# B&R Automation Studio project Panasonic_LinkaPowerCP2_A2021055 (part 28)

#### Main.st - Init, cyclic, exit code
```iecst
PROGRAM _INIT
	(* Insert code here *)

END_PROGRAM

PROGRAM _CYCLIC

	//Volanie funkcie SequenceControl//
	SequenceControl(SC:= SC_P3_ZdvizkaPredLeakTestA);

	//Volanie podprogramov//
	OvlZdvizky;

	//Reset sekcie //
	IF P3_ZdvizkaPredLeakTestA.Reset THEN
		SC_P3_ZdvizkaPredLeakTestA.Step:= 0;
		P3_ZdvizkaPredLeakTestA.Reset:= FALSE;
	ELSIF NOT Safety.STAV.Linka_ZonaCS_AKTIVNA THEN
		SC_P3_ZdvizkaPredLeakTestA.Step:= 0;
	END_IF

	CASE SC_P3_ZdvizkaPredLeakTestA.Step OF

		0:
			SC_P3_ZdvizkaPredLeakTestA.StepName:='0 - Nulovanie';
			SC_OvlZdvizky.Step:= 0;
			P3_ZdvizkaPredLeakTestA.Automat:= FALSE;
			P3_ZdvizkaPredLeakTestA.KoniecCyklu:= FALSE;
			P3_ZdvizkaPredLeakTestA.Manual:= FALSE;
			P3_ZdvizkaPredLeakTestA.STAV.PoINIT:= FALSE;
			P3_ZdvizkaPredLeakTestA.OUT.TlmicPaletky_VYSUN:= FALSE;
			P3_Dopravniky.OUT.PriecnyDopravnik1_VPRED:= FALSE;
			P3_ZdvizkaPredLeakTestA.STAV.PrebiehaVyvezeniePaletkyNaTratA:= FALSE;
			P3_ZdvizkaPredLeakTestA.STAV.PrebiehaVyvezeniePaletkyNaTratB:= FALSE;
			P3_HV_Test.STAV.PrebiehaVyvezeniePaletky:= FALSE;

			IF Safety.STAV.Linka_ZonaCS_AKTIVNA AND
				Safety.STAV.P3_ZonaBunky_AKTIVNA AND
				P3_Pracovisko.STAV.HardwareBunky_OK AND
				NOT P3_Pracovisko.STAV.Porucha_ST1 AND
				NOT P3_Pracovisko.STAV.Porucha_ST2 AND
				NOT P3_Pracovisko.STAV.Porucha_ST3 AND
				NOT P3_Pracovisko.STAV.Porucha_ST4 AND
				NOT P3_Pracovisko.STAV.Porucha_ST5 AND
				NOT P3_Pracovisko.STAV.Porucha_ST6 AND
				NOT P3_Pracovisko.STAV.Porucha_ST7 AND
				NOT P3_Pracovisko.STAV.Porucha_ST8 THEN
				SC_P3_ZdvizkaPredLeakTestA.ResetStep:= TRUE;
				SC_P3_ZdvizkaPredLeakTestA.Step:= 1;
			END_IF

		1:
			SC_P3_ZdvizkaPredLeakTestA.StepName:='1 - Cakam na spustenie vyroby';
			P3_ZdvizkaPredLeakTestA.KoniecCyklu:= FALSE;
			IF P3_ZdvizkaPredLeakTestA.Automat THEN
				SC_P3_ZdvizkaPredLeakTestA.Step:= 2;
			ELSIF P3_ZdvizkaPredLeakTestA.Manual THEN
				SC_P3_ZdvizkaPredLeakTestA.Step:= 700;
			END_IF

			//********************************************************Inicializácia****************************************************************************//

		2:
			SC_P3_ZdvizkaPredLeakTestA.StepName:='2 - Inicializacia - cakam na spustenie inicializacie';
			SC_P3_ZdvizkaPredLeakTestA.IdleTime.PT:= T#500ms;
			SC_P3_ZdvizkaPredLeakTestA.AlarmTime.PT:= T#5s;

			IF P3_Dopravniky.STAV.PoINIT AND P3_ZdvizkaPredLeakTestB.STAV.PoINIT THEN
				SC_P3_ZdvizkaPredLeakTestA.ResetStep:= TRUE;
				SC_P3_ZdvizkaPredLeakTestA.Step:= 5;
			END_IF

		5:
			SC_P3_ZdvizkaPredLeakTestA.StepName:='5 - Inicializacia - kontrola pozicie zdvizky';
			SC_P3_ZdvizkaPredLeakTestA.IdleTime.PT:= T#500ms;
			SC_P3_ZdvizkaPredLeakTestA.AlarmTime.PT:= T#5s;

			IF P3_ZdvizkaPredLeakTestA.IN.Zdvizka_StrednaPoloha AND P3_ZdvizkaPredLeakTestA.IN.PritomnostPaletky THEN
				P3_ZdvizkaPredLeakTestA.STAV.PoINIT:= TRUE;
				SC_P3_ZdvizkaPredLeakTestA.ResetStep:= TRUE;
				SC_P3_ZdvizkaPredLeakTestA.Step:= 100;
			ELSIF P3_ZdvizkaPredLeakTestA.IN.Zdvizka_StrednaPoloha AND NOT P3_ZdvizkaPredLeakTestA.IN.PritomnostPaletky THEN
				SC_P3_ZdvizkaPredLeakTestA.ResetStep:= TRUE;
				SC_P3_ZdvizkaPredLeakTestA.Step:= 6;
			ELSE
				SC_P3_ZdvizkaPredLeakTestA.ResetStep:= TRUE;
				SC_P3_ZdvizkaPredLeakTestA.Step:= 8;
			END_IF

		6:
			SC_P3_ZdvizkaPredLeakTestA.StepName:='5 - Inicializacia - vysunutie tlmica';
			SC_P3_ZdvizkaPredLeakTestA.IdleTime.PT:= T#500ms;
			SC_P3_ZdvizkaPredLeakTestA.AlarmTime.PT:= T#5s;

			IF NOT SC_P3_ZdvizkaPredLeakTestA.Switch1 THEN
				P3_ZdvizkaPredLeakTestA.OUT.TlmicPaletky_VYSUN:= TRUE;
				SC_P3_ZdvizkaPredLeakTestA.IdleTime.IN:= TRUE;
				SC_P3_ZdvizkaPredLeakTestA.Switch1:= TRUE;
			END_IF

			IF SC_P3_ZdvizkaPredLeakTestA.IdleTime.Q THEN
				P3_ZdvizkaPredLeakTestA.OUT.TlmicPaletky_VYSUN:= FALSE;
				P3_ZdvizkaPredLeakTestA.STAV.PoINIT:= TRUE;
				SC_P3_ZdvizkaPredLeakTestA.ResetStep:= TRUE;
				SC_P3_ZdvizkaPredLeakTestA.Step:= 100;
			END_IF

		8:
			SC_P3_ZdvizkaPredLeakTestA.StepName:='8 - Inicializacia - presun zdvizky do strednej polohy';
			SC_P3_ZdvizkaPredLeakTestA.IdleTime.PT:= T#5s;
			SC_P3_ZdvizkaPredLeakTestA.AlarmTime.PT:= T#5s;

			IF NOT SC_P3_ZdvizkaPredLeakTestA.Switch1 AND SC_OvlZdvizky.Step = 1 THEN
				Zdvizku_VYSTRED:= TRUE;
				SC_P3_ZdvizkaPredLeakTestA.Switch1:= TRUE;
			END_IF

			IF P3_ZdvizkaPredLeakTestA.IN.Zdvizka_StrednaPoloha THEN
				SC_P3_ZdvizkaPredLeakTestA.ResetStep:= TRUE;
				SC_P3_ZdvizkaPredLeakTestA.Step:= 10;
			END_IF

		10:
			SC_P3_ZdvizkaPredLeakTestA.StepName:='10 - Inicializacia - hladania paletky';
			SC_P3_ZdvizkaPredLeakTestA.IdleTime.PT:= T#5s;
			SC_P3_ZdvizkaPredLeakTestA.AlarmTime.PT:= T#5s;

			SC_P3_ZdvizkaPredLeakTestA.IdleTime.IN:= TRUE;

			IF SC_P3_ZdvizkaPredLeakTestA.IdleTime.Q THEN
				SC_P3_ZdvizkaPredLeakTestA.ResetStep:= TRUE;
				SC_P3_ZdvizkaPredLeakTestA.Step:= 5;
			END_IF

			//********************************************************Automatický režim****************************************************************************//

		100:
			SC_P3_ZdvizkaPredLeakTestA.StepName:='100 - Automaticky Rezim - cakam na príchod paletky na zdvizku';
			SC_P3_ZdvizkaPredLeakTestA.IdleTime.PT:= T#700ms;
			SC_P3_ZdvizkaPredLeakTestA.AlarmTime.PT:= T#5s;

			SC_P3_ZdvizkaPredLeakTestA.IdleTime.IN:= P3_ZdvizkaPredLeakTestA.IN.PritomnostPaletky;

			IF P3_ZdvizkaPredLeakTestA.IN.PritomnostPaletky THEN
				P3_HV_Test.STAV.PrebiehaVyvezeniePaletky:= FALSE;
			END_IF

			IF P3_ZdvizkaPredLeakTestA.KoniecCyklu AND NOT P3_HV_Test.Automat THEN
				SC_P3_ZdvizkaPredLeakTestA.ResetStep:= TRUE;
				SC_P3_ZdvizkaPredLeakTestA.Step:= 0;
			ELSIF SC_P3_ZdvizkaPredLeakTestA.IdleTime.Q THEN
				SC_P3_ZdvizkaPredLeakTestA.ResetStep:= TRUE;
				SC_P3_ZdvizkaPredLeakTestA.Step:= 101;
			END_IF

		101:
			SC_P3_ZdvizkaPredLeakTestA.StepName:='101 - Automaticky Rezim - rozhodnutie o smere vyvazania';
			SC_P3_ZdvizkaPredLeakTestA.IdleTime.PT:= T#200ms;
			SC_P3_ZdvizkaPredLeakTestA.AlarmTime.PT:= T#5s;

			IF P3_ZdvizkaPredLeakTestA.KoniecCyklu AND NOT P3_HV_Test.Automat THEN
				SC_P3_ZdvizkaPredLeakTestA.ResetStep:= TRUE;
				SC_P3_ZdvizkaPredLeakTestA.Step:= 0;
			ELSIF P3_LeakageTestA.STAV.Tester_ON AND NOT P3_LeakageTestA.RFID_hlava.PritomnostPaletky AND SC_P3_LeakageTestA.Step = 100 AND NOT P3_ZdvizkaPredLeakTestA.STAV.PrebiehaVyvezeniePaletkyNaTratA THEN
				SC_P3_ZdvizkaPredLeakTestA.ResetStep:= TRUE;
				SC_P3_ZdvizkaPredLeakTestA.Step:= 110;
			ELSIF P3_LeakageTestB.STAV.Tester_ON AND NOT P3_ZdvizkaPredLeakTestB.IN.PritomnostPaletky AND NOT P3_LeakageTestB.RFID_hlava.PritomnostPaletky AND SC_P3_ZdvizkaPredLeakTestB.Step = 100 AND NOT P3_ZdvizkaPredLeakTestA.STAV.PrebiehaVyvezeniePaletkyNaTratB THEN
				SC_P3_ZdvizkaPredLeakTestA.ResetStep:= TRUE;
				SC_P3_ZdvizkaPredLeakTestA.Step:= 120;
			END_IF

			//Vyvážanie na trať A//

		110:
			SC_P3_ZdvizkaPredLeakTestA.StepName:='110 - Automaticky Rezim - presun zdvizky do spodnej polohy';
			SC_P3_ZdvizkaPredLeakTestA.IdleTime.PT:= T#200ms;
			SC_P3_ZdvizkaPredLeakTestA.AlarmTime.PT:= T#5s;

			IF NOT SC_P3_ZdvizkaPredLeakTestA.Switch1 AND SC_OvlZdvizky.Step = 1 THEN
				Zdvizku_ZASUN:= TRUE;
				P3_ZdvizkaPredLeakTestA.STAV.PrebiehaVyvezeniePaletkyNaTratA:= TRUE;
				SC_P3_ZdvizkaPredLeakTestA.Switch1:= TRUE;
			END_IF

			IF P3_ZdvizkaPredLeakTestA.IN.Zdvizka_SpodnaPoloha THEN
				SC_P3_ZdvizkaPredLeakTestA.ResetStep:= TRUE;
				SC_P3_ZdvizkaPredLeakTestA.Step:= 113;
			END_IF

		113:
			SC_P3_ZdvizkaPredLeakTestA.StepName:='113 - Automaticky Rezim - cakam na ukoncenie vyvazania na Trat A';
			SC_P3_ZdvizkaPredLeakTestA.IdleTime.PT:= T#500ms;
			SC_P3_ZdvizkaPredLeakTestA.AlarmTime.PT:= T#5s;

			IF P3_LeakageTestA.RFID_hlava.PritomnostPaletky AND SC_OvlZdvizky.Step = 1 AND NOT SC_P3_ZdvizkaPredLeakTestA.Switch1 THEN
				Zdvizku_VYSTRED:= TRUE;
				SC_P3_ZdvizkaPredLeakTestA.Switch1:= TRUE;
			END_IF

			IF P3_ZdvizkaPredLeakTestA.IN.Zdvizka_StrednaPoloha THEN
				SC_P3_ZdvizkaPredLeakTestA.ResetStep:= TRUE;
				SC_P3_ZdvizkaPredLeakTestA.Step:= 130;
			END_IF

			//Vyvážanie na trať B//

		120:
			SC_P3_ZdvizkaPredLeakTestA.StepName:='120 - Automaticky Rezim - presun zdviziek do hornej polohy';
			SC_P3_ZdvizkaPredLeakTestA.IdleTime.PT:= T#200ms;
			SC_P3_ZdvizkaPredLeakTestA.AlarmTime.PT:= T#5s;

			IF NOT SC_P3_ZdvizkaPredLeakTestA.Switch1 AND SC_OvlZdvizky.Step = 1 THEN
				Zdvizku_VYSUN:= TRUE;
				P3_ZdvizkaPredLeakTestB.OUT.Zdvizku_ZASUN:= FALSE;
				P3_ZdvizkaPredLeakTestB.OUT.Zdvizku_VYSUN:= TRUE;
				P3_ZdvizkaPredLeakTestA.STAV.PrebiehaVyvezeniePaletkyNaTratB:= TRUE;
				SC_P3_ZdvizkaPredLeakTestA.Switch1:= TRUE;
			END_IF

			IF P3_ZdvizkaPredLeakTestA.IN.Zdvizka_HornaPoloha AND P3_ZdvizkaPredLeakTestB.IN.Zdvizka_HornaPoloha THEN
				SC_P3_ZdvizkaPredLeakTestA.ResetStep:= TRUE;
				SC_P3_ZdvizkaPredLeakTestA.Step:= 123;
			END_IF

		123:
			SC_P3_ZdvizkaPredLeakTestA.StepName:='123 - Automaticky Rezim - cakam na ukoncenie vyvazania na Trat B';
			SC_P3_ZdvizkaPredLeakTestA.IdleTime.PT:= T#500ms;
			SC_P3_ZdvizkaPredLeakTestA.AlarmTime.PT:= T#5s;

			SC_P3_ZdvizkaPredLeakTestA.IdleTime.IN:= P3_ZdvizkaPredLeakTestB.IN.PritomnostPaletky;

			IF NOT SC_P3_ZdvizkaPredLeakTestA.Switch1 THEN
				P3_Dopravniky.OUT.PriecnyDopravnik1_VPRED:= TRUE;
				SC_P3_ZdvizkaPredLeakTestA.Switch1:= TRUE;
			END_IF

			IF SC_P3_ZdvizkaPredLeakTestA.IdleTime.Q THEN
				P3_Dopravniky.OUT.PriecnyDopravnik1_VPRED:= FALSE;
				SC_P3_ZdvizkaPredLeakTestA.ResetStep:= TRUE;
				SC_P3_ZdvizkaPredLeakTestA.Step:= 125;
			END_IF

		125:
			SC_P3_ZdvizkaPredLeakTestA.StepName:='123 - Automaticky Rezim - cakam na presun zdviziek do strednej polohy';
			SC_P3_ZdvizkaPredLeakTestA.IdleTime.PT:= T#1s;
			SC_P3_ZdvizkaPredLeakTestA.AlarmTime.PT:= T#5s;

			IF NOT SC_P3_ZdvizkaPredLeakTestA.Switch1 AND SC_OvlZdvizky.Step = 1 THEN
				Zdvizku_VYSTRED:= TRUE;
				P3_ZdvizkaPredLeakTestB.OUT.Zdvizku_ZASUN:= FALSE;
				P3_ZdvizkaPredLeakTestB.OUT.Zdvizku_VYSUN:= FALSE;
				SC_P3_ZdvizkaPredLeakTestA.Switch1:= TRUE;
			END_IF

			IF P3_ZdvizkaPredLeakTestA.IN.Zdvizka_StrednaPoloha AND P3_ZdvizkaPredLeakTestB.IN.Zdvizka_StrednaPoloha THEN
				P3_ZdvizkaPredLeakTestA.STAV.PrebiehaVyvezeniePaletkyNaTratB:= FALSE;
				SC_P3_ZdvizkaPredLeakTestA.ResetStep:= TRUE;
				SC_P3_ZdvizkaPredLeakTestA.Step:= 130;
			END_IF

			//Vysunutie tlmenia paletky//

		130:
			SC_P3_ZdvizkaPredLeakTestA.StepName:='130 - Automaticky Rezim - vysunutie tlamena paletky';
			SC_P3_ZdvizkaPredLeakTestA.IdleTime.PT:= T#1s;
			SC_P3_ZdvizkaPredLeakTestA.AlarmTime.PT:= T#5s;

			IF NOT SC_P3_ZdvizkaPredLeakTestA.Switch1 THEN
				P3_ZdvizkaPredLeakTestA.OUT.TlmicPaletky_VYSUN:= TRUE;
				SC_P3_ZdvizkaPredLeakTestA.IdleTime.IN:= TRUE;
				SC_P3_ZdvizkaPredLeakTestA.Switch1:= TRUE;
			END_IF

			IF SC_P3_ZdvizkaPredLeakTestA.IdleTime.Q THEN
				P3_ZdvizkaPredLeakTestA.OUT.TlmicPaletky_VYSUN:= FALSE;
				SC_P3_ZdvizkaPredLeakTestA.ResetStep:= TRUE;
				SC_P3_ZdvizkaPredLeakTestA.Step:= 100;
			END_IF

			//*******************************************************Manuálny režim*******************************************************************************//
		700:
			SC_P3_ZdvizkaPredLeakTestA.StepName:='700 - Manualny Rezim';
			SC_P3_ZdvizkaPredLeakTestA.IdleTime.PT:= T#8s;
			SC_P3_ZdvizkaPredLeakTestA.AlarmTime.PT:= T#5s;

	END_CASE

				END_PROGRAM

PROGRAM _EXIT
				(* Insert code here *)

				END_PROGRAM
```

#### Variables.var - Local variables
```iecst
VAR
	SC_OvlZdvizky : SequenceControlTyp;
	Zdvizku_VYSUN : BOOL;
	Zdvizku_ZASUN : BOOL;
	Zdvizku_VYSTRED : BOOL := FALSE;
END_VAR
```

#### OvlZdvizky.st
```iecst
ACTION OvlZdvizky:

	//Volanie funkcie SequenceControl//
	SequenceControl(SC:= SC_OvlZdvizky);

	CASE SC_OvlZdvizky.Step OF

		0:
			SC_OvlZdvizky.StepName:= '0 - Nulovanie';
			Zdvizku_VYSUN:= FALSE;
			Zdvizku_ZASUN:= FALSE;
			Zdvizku_VYSTRED:= FALSE;

			IF SC_P3_ZdvizkaPredLeakTestA.Step <> 0 THEN
				SC_OvlZdvizky.ResetStep:= TRUE;
				SC_OvlZdvizky.Step:= 1;
			END_IF

		1:
			SC_OvlZdvizky.StepName:= '1 - Rozhodnutie o cinnosti';
			IF Zdvizku_VYSUN THEN
				SC_OvlZdvizky.Step:= 10;
			ELSIF Zdvizku_ZASUN THEN
				SC_OvlZdvizky.Step:= 20;
			ELSIF Zdvizku_VYSTRED THEN
				SC_OvlZdvizky.Step:= 30;
			END_IF

		10:
			SC_OvlZdvizky.StepName:= '10 - Vysunutie zdvizky hore';
			SC_OvlZdvizky.IdleTime.PT:= T#3s;
			SC_OvlZdvizky.AlarmTime.PT:= T#6s;

			IF P3_ZdvizkaPredLeakTestA.Automat THEN
				SC_OvlZdvizky.AlarmTime.IN:= TRUE;
			ELSE
				SC_OvlZdvizky.IdleTime.IN:= TRUE;
			END_IF

			IF NOT SC_OvlZdvizky.Switch1 THEN
				P3_ZdvizkaPredLeakTestA.OUT.Zdvizku_ZASUN:= FALSE;
				P3_ZdvizkaPredLeakTestA.OUT.Zdvizku_VYSUN:= TRUE;
				SC_OvlZdvizky.Switch1:= TRUE;
			END_IF

			IF P3_ZdvizkaPredLeakTestA.IN.Zdvizka_HornaPoloha OR SC_OvlZdvizky.IdleTime.Q THEN
				SC_OvlZdvizky.ResetStep:= TRUE;
				SC_OvlZdvizky.Step:= 0;
			ELSIF SC_OvlZdvizky.AlarmTime.Q THEN
				P34_Alarmy[368]:= TRUE;
				P3_Pracovisko.STAV.Porucha_ST3:= TRUE;
			END_IF

		20:
			SC_OvlZdvizky.StepName:= '20 - Zasunutie zdvizky dole';
			SC_OvlZdvizky.IdleTime.PT:= T#3s;
			SC_OvlZdvizky.AlarmTime.PT:= T#6s;

			IF P3_ZdvizkaPredLeakTestA.Automat THEN
				SC_OvlZdvizky.AlarmTime.IN:= TRUE;
			ELSE
				SC_OvlZdvizky.IdleTime.IN:= TRUE;
			END_IF

			IF NOT SC_OvlZdvizky.Switch1 THEN
				P3_ZdvizkaPredLeakTestA.OUT.Zdvizku_VYSUN:= FALSE;
				P3_ZdvizkaPredLeakTestA.OUT.Zdvizku_ZASUN:= TRUE;
				SC_OvlZdvizky.Switch1:= TRUE;
			END_IF

			IF P3_ZdvizkaPredLeakTestA.IN.Zdvizka_SpodnaPoloha OR SC_OvlZdvizky.IdleTime.Q THEN
				SC_OvlZdvizky.ResetStep:= TRUE;
				SC_OvlZdvizky.Step:= 0;
			ELSIF SC_OvlZdvizky.AlarmTime.Q THEN
				P34_Alarmy[369]:= TRUE;
				P3_Pracovisko.STAV.Porucha_ST3:= TRUE;
			END_IF

		30:
			SC_OvlZdvizky.StepName:= '30 - Presun zdvizky do strednej polohy';
			SC_OvlZdvizky.IdleTime.PT:= T#3s;
			SC_OvlZdvizky.AlarmTime.PT:= T#6s;

			IF P3_ZdvizkaPredLeakTestA.Automat THEN
				SC_OvlZdvizky.AlarmTime.IN:= TRUE;
			ELSE
				SC_OvlZdvizky.IdleTime.IN:= TRUE;
			END_IF

			IF NOT SC_OvlZdvizky.Switch1 THEN
				P3_ZdvizkaPredLeakTestA.OUT.Zdvizku_VYSUN:= FALSE;
				P3_ZdvizkaPredLeakTestA.OUT.Zdvizku_ZASUN:= FALSE;
				SC_OvlZdvizky.Switch1:= TRUE;
			END_IF

			IF P3_ZdvizkaPredLeakTestA.IN.Zdvizka_StrednaPoloha OR SC_OvlZdvizky.IdleTime.Q THEN
				SC_OvlZdvizky.ResetStep:= TRUE;
				SC_OvlZdvizky.Step:= 0;
			ELSIF SC_OvlZdvizky.AlarmTime.Q THEN
				P34_Alarmy[370]:= TRUE;
				P3_Pracovisko.STAV.Porucha_ST3:= TRUE;
			END_IF

	END_CASE

END_ACTION
```

### Program Logical/Program/Pracovisko_3/P3_ZdvizkaPredLeakTestB (IEC)

#### Main.st - Init, cyclic, exit code
```iecst
PROGRAM _INIT
	(* Insert code here *)

END_PROGRAM

PROGRAM _CYCLIC

	//Volanie funkcie SequenceControl//
	SequenceControl(SC:= SC_P3_ZdvizkaPredLeakTestB);

	//Volanie podprogramov//
	OvlZdvizky;

	//Reset sekcie //
	IF P3_ZdvizkaPredLeakTestB.Reset THEN
		SC_P3_ZdvizkaPredLeakTestB.Step:= 0;
		P3_ZdvizkaPredLeakTestB.Reset:= FALSE;
	ELSIF NOT Safety.STAV.Linka_ZonaCS_AKTIVNA THEN
		SC_P3_ZdvizkaPredLeakTestB.Step:= 0;
	END_IF

	CASE SC_P3_ZdvizkaPredLeakTestB.Step OF

		0:
			SC_P3_ZdvizkaPredLeakTestB.StepName:='0 - Nulovanie';
			SC_OvlZdvizky.Step:= 0;
			P3_ZdvizkaPredLeakTestB.Automat:= FALSE;
			P3_ZdvizkaPredLeakTestB.KoniecCyklu:= FALSE;
			P3_ZdvizkaPredLeakTestB.Manual:= FALSE;
			P3_ZdvizkaPredLeakTestB.STAV.PoINIT:= FALSE;
			P3_Dopravniky.OUT.PriecnyDopravnik1_VPRED:= FALSE;
			P3_ZdvizkaPredLeakTestB.STAV.PrebiehaVyvezeniePaletky:= FALSE;
			P3_ZdvizkaPredLeakTestA.STAV.PrebiehaVyvezeniePaletkyNaTratB:= FALSE;

			IF Safety.STAV.Linka_ZonaCS_AKTIVNA AND
				Safety.STAV.P3_ZonaBunky_AKTIVNA AND
				P3_Pracovisko.STAV.HardwareBunky_OK AND
				NOT P3_Pracovisko.STAV.Porucha_ST1 AND
				NOT P3_Pracovisko.STAV.Porucha_ST2 AND
				NOT P3_Pracovisko.STAV.Porucha_ST3 AND
				NOT P3_Pracovisko.STAV.Porucha_ST4 AND
				NOT P3_Pracovisko.STAV.Porucha_ST5 AND
				NOT P3_Pracovisko.STAV.Porucha_ST6 AND
				NOT P3_Pracovisko.STAV.Porucha_ST7 AND
				NOT P3_Pracovisko.STAV.Porucha_ST8 THEN
				SC_P3_ZdvizkaPredLeakTestB.ResetStep:= TRUE;
				SC_P3_ZdvizkaPredLeakTestB.Step:= 1;
			END_IF

		1:
			SC_P3_ZdvizkaPredLeakTestB.StepName:='1 - Cakam na spustenie vyroby';
			P3_ZdvizkaPredLeakTestB.KoniecCyklu:= FALSE;
			IF P3_ZdvizkaPredLeakTestB.Automat THEN
				SC_P3_ZdvizkaPredLeakTestB.Step:= 2;
			ELSIF P3_ZdvizkaPredLeakTestB.Manual THEN
				SC_P3_ZdvizkaPredLeakTestB.Step:= 700;
			END_IF

			//********************************************************Inicializácia****************************************************************************//

		2:
			SC_P3_ZdvizkaPredLeakTestB.StepName:='2 - Inicializacia - cakam na spustenie inicializacie';
			SC_P3_ZdvizkaPredLeakTestB.IdleTime.PT:= T#500ms;
			SC_P3_ZdvizkaPredLeakTestB.AlarmTime.PT:= T#5s;

			IF P3_Dopravniky.STAV.PoINIT THEN
				SC_P3_ZdvizkaPredLeakTestB.ResetStep:= TRUE;
				SC_P3_ZdvizkaPredLeakTestB.Step:= 5;
			END_IF

		5:
			SC_P3_ZdvizkaPredLeakTestB.StepName:='5 - Inicializacia - kontrola pozicie zdvizky';
			SC_P3_ZdvizkaPredLeakTestB.IdleTime.PT:= T#500ms;
			SC_P3_ZdvizkaPredLeakTestB.AlarmTime.PT:= T#5s;

			IF P3_ZdvizkaPredLeakTestB.IN.Zdvizka_StrednaPoloha AND P3_ZdvizkaPredLeakTestB.IN.PritomnostPaletky THEN
				P3_ZdvizkaPredLeakTestB.STAV.PoINIT:= TRUE;
				SC_P3_ZdvizkaPredLeakTestB.ResetStep:= TRUE;
				SC_P3_ZdvizkaPredLeakTestB.Step:= 120;
			ELSE
				SC_P3_ZdvizkaPredLeakTestB.ResetStep:= TRUE;
				SC_P3_ZdvizkaPredLeakTestB.Step:= 8;
			END_IF

		8:
			SC_P3_ZdvizkaPredLeakTestB.StepName:='8 - Inicializacia - presun zdvizky do hornej polohy';
			SC_P3_ZdvizkaPredLeakTestB.IdleTime.PT:= T#500ms;
			SC_P3_ZdvizkaPredLeakTestB.AlarmTime.PT:= T#5s;

			IF NOT SC_P3_ZdvizkaPredLeakTestB.Switch1 AND SC_OvlZdvizky.Step = 1 THEN
				Zdvizku_VYSUN:= TRUE;
				SC_P3_ZdvizkaPredLeakTestB.Switch1:= TRUE;
			END_IF

			IF P3_ZdvizkaPredLeakTestB.IN.Zdvizka_HornaPoloha THEN
				SC_P3_ZdvizkaPredLeakTestB.ResetStep:= TRUE;
				SC_P3_ZdvizkaPredLeakTestB.Step:= 10;
			END_IF

		10:
			SC_P3_ZdvizkaPredLeakTestB.StepName:='10 - Inicializacia - kontrola pritomnosti paletky na zdvizke pred Leakage Testom A';
			SC_P3_ZdvizkaPredLeakTestB.IdleTime.PT:= T#500ms;
			SC_P3_ZdvizkaPredLeakTestB.AlarmTime.PT:= T#5s;

			IF NOT P3_ZdvizkaPredLeakTestA.IN.PritomnostPaletky THEN
				P3_ZdvizkaPredLeakTestA.OUT.Zdvizku_ZASUN:= FALSE;
				P3_ZdvizkaPredLeakTestA.OUT.Zdvizku_VYSUN:= TRUE;
				SC_P3_ZdvizkaPredLeakTestB.ResetStep:= TRUE;
				SC_P3_ZdvizkaPredLeakTestB.Step:= 11;
			ELSE
				SC_P3_ZdvizkaPredLeakTestB.ResetStep:= TRUE;
				SC_P3_ZdvizkaPredLeakTestB.Step:= 13;
			END_IF

		11:
			SC_P3_ZdvizkaPredLeakTestB.StepName:='11 - Inicializacia - cakam na zodvihnutie zdvizky Pred Leakage Testom A';
			SC_P3_ZdvizkaPredLeakTestB.IdleTime.PT:= T#500ms;
			SC_P3_ZdvizkaPredLeakTestB.AlarmTime.PT:= T#5s;

			IF P3_ZdvizkaPredLeakTestA.IN.Zdvizka_HornaPoloha THEN
				SC_P3_ZdvizkaPredLeakTestB.ResetStep:= TRUE;
				SC_P3_ZdvizkaPredLeakTestB.Step:= 13;
			END_IF

		13:
			SC_P3_ZdvizkaPredLeakTestB.StepName:='13 - Inicializacia - spustenie priecneho dopravnika';
			SC_P3_ZdvizkaPredLeakTestB.IdleTime.PT:= T#500ms;
			SC_P3_ZdvizkaPredLeakTestB.AlarmTime.PT:= T#7s;

			SC_P3_ZdvizkaPredLeakTestB.IdleTime.IN:= P3_ZdvizkaPredLeakTestB.IN.PritomnostPaletky AND P3_ZdvizkaPredLeakTestB.IN.PoziciaPaletky_OK;

			IF NOT SC_P3_ZdvizkaPredLeakTestB.Switch1 THEN
				P3_Dopravniky.OUT.PriecnyDopravnik1_VPRED:= TRUE;
				SC_P3_ZdvizkaPredLeakTestB.AlarmTime.IN:= TRUE;
				SC_P3_ZdvizkaPredLeakTestB.Switch1:= TRUE;
			END_IF

			IF SC_P3_ZdvizkaPredLeakTestB.IdleTime.Q THEN
				P3_Dopravniky.OUT.PriecnyDopravnik1_VPRED:= FALSE;
				SC_P3_ZdvizkaPredLeakTestB.ResetStep:= TRUE;
				SC_P3_ZdvizkaPredLeakTestB.Step:= 15;
			ELSIF SC_P3_ZdvizkaPredLeakTestB.AlarmTime.Q THEN
				P3_Dopravniky.OUT.PriecnyDopravnik1_VPRED:= FALSE;
				SC_P3_ZdvizkaPredLeakTestB.ResetStep:= TRUE;
				SC_P3_ZdvizkaPredLeakTestB.Step:= 15;
			END_IF

		15:
			SC_P3_ZdvizkaPredLeakTestB.StepName:='15 - Inicializacia - presun zdvizky do strednej polohy';
			SC_P3_ZdvizkaPredLeakTestB.IdleTime.PT:= T#500ms;
			SC_P3_ZdvizkaPredLeakTestB.AlarmTime.PT:= T#5s;

			IF NOT SC_P3_ZdvizkaPredLeakTestB.Switch1 AND SC_OvlZdvizky.Step = 1 THEN
				Zdvizku_VYSTRED:= TRUE;
				P3_ZdvizkaPredLeakTestA.OUT.Zdvizku_ZASUN:= FALSE;
				P3_ZdvizkaPredLeakTestA.OUT.Zdvizku_VYSUN:= FALSE;
				SC_P3_ZdvizkaPredLeakTestB.Switch1:= TRUE;
			END_IF

			IF P3_ZdvizkaPredLeakTestB.IN.Zdvizka_StrednaPoloha AND P3_ZdvizkaPredLeakTestA.IN.Zdvizka_StrednaPoloha THEN
				P3_ZdvizkaPredLeakTestB.STAV.PoINIT:= TRUE;
				IF P3_ZdvizkaPredLeakTestB.IN.PritomnostPaletky THEN
					SC_P3_ZdvizkaPredLeakTestB.ResetStep:= TRUE;
					SC_P3_ZdvizkaPredLeakTestB.Step:= 120;
				ELSE
					SC_P3_ZdvizkaPredLeakTestB.ResetStep:= TRUE;
					SC_P3_ZdvizkaPredLeakTestB.Step:= 100;
				END_IF
			END_IF

		//********************************************************Automatický režim****************************************************************************//
		100:
			SC_P3_ZdvizkaPredLeakTestB.StepName:='100 - Automaticky Rezim - cakam na prichod paletky na zdvizku';
			SC_P3_ZdvizkaPredLeakTestB.IdleTime.PT:= T#200ms;
			SC_P3_ZdvizkaPredLeakTestB.AlarmTime.PT:= T#5s;

			SC_P3_ZdvizkaPredLeakTestB.IdleTime.IN:= P3_ZdvizkaPredLeakTestB.IN.PritomnostPaletky AND P3_ZdvizkaPredLeakTestB.IN.Zdvizka_StrednaPoloha;

			IF P3_ZdvizkaPredLeakTestB.IN.PritomnostPaletky THEN
				P3_ZdvizkaPredLeakTestA.STAV.PrebiehaVyvezeniePaletkyNaTratB:= FALSE;
			END_IF

			IF P3_ZdvizkaPredLeakTestB.KoniecCyklu AND NOT P3_ZdvizkaPredLeakTestA.Automat THEN
				SC_P3_ZdvizkaPredLeakTestB.ResetStep:= TRUE;
				SC_P3_ZdvizkaPredLeakTestB.Step:= 0;
			ELSIF SC_P3_ZdvizkaPredLeakTestB.IdleTime.Q THEN
				SC_P3_ZdvizkaPredLeakTestB.ResetStep:= TRUE;
				SC_P3_ZdvizkaPredLeakTestB.Step:= 120;
			END_IF

		120:
			SC_P3_ZdvizkaPredLeakTestB.StepName:='120 - Automaticky Rezim - cakam na vyvezenie na stoper Leakage Testu B';
			SC_P3_ZdvizkaPredLeakTestB.IdleTime.PT:= T#500ms;
			SC_P3_ZdvizkaPredLeakTestB.AlarmTime.PT:= T#5s;

			IF P3_ZdvizkaPredLeakTestB.KoniecCyklu AND NOT P3_ZdvizkaPredLeakTestA.Automat THEN
				SC_P3_ZdvizkaPredLeakTestB.ResetStep:= TRUE;
				SC_P3_ZdvizkaPredLeakTestB.Step:= 0;
			ELSIF NOT P3_LeakageTestB.RFID_hlava.PritomnostPaletky AND SC_P3_LeakageTestB.Step = 100 THEN
				SC_P3_ZdvizkaPredLeakTestB.ResetStep:= TRUE;
				SC_P3_ZdvizkaPredLeakTestB.Step:= 123;
			END_IF

		123:
			SC_P3_ZdvizkaPredLeakTestB.StepName:='123 - Automaticky Rezim - presun zdvizky do spodnej polohy';
			SC_P3_ZdvizkaPredLeakTestB.IdleTime.PT:= T#200ms;
			SC_P3_ZdvizkaPredLeakTestB.AlarmTime.PT:= T#5s;

			IF NOT SC_P3_ZdvizkaPredLeakTestB.Switch1 AND SC_OvlZdvizky.Step = 1 THEN
				Zdvizku_ZASUN:= TRUE;
				P3_ZdvizkaPredLeakTestB.STAV.PrebiehaVyvezeniePaletky:= TRUE;
				SC_P3_ZdvizkaPredLeakTestB.Switch1:= TRUE;
			END_IF

			IF P3_ZdvizkaPredLeakTestB.IN.Zdvizka_SpodnaPoloha THEN
				SC_P3_ZdvizkaPredLeakTestB.ResetStep:= TRUE;
				SC_P3_ZdvizkaPredLeakTestB.Step:= 125;
			END_IF

		125:
			SC_P3_ZdvizkaPredLeakTestB.StepName:='125 - Automaticky Rezim - cakam na ukoncenie vyvazania na stoper Leakage Testu B';
			SC_P3_ZdvizkaPredLeakTestB.IdleTime.PT:= T#500ms;
			SC_P3_ZdvizkaPredLeakTestB.AlarmTime.PT:= T#5s;

			IF P3_LeakageTestB.RFID_hlava.PritomnostPaletky AND NOT SC_P3_ZdvizkaPredLeakTestB.Switch1 AND SC_OvlZdvizky.Step = 1 THEN
				Zdvizku_VYSTRED:= TRUE;
				SC_P3_ZdvizkaPredLeakTestB.Switch1:= TRUE;
			END_IF

			IF P3_ZdvizkaPredLeakTestB.IN.Zdvizka_StrednaPoloha THEN
				SC_P3_ZdvizkaPredLeakTestB.ResetStep:= TRUE;
				SC_P3_ZdvizkaPredLeakTestB.Step:= 100;
			END_IF

			//*******************************************************Manuálny režim*******************************************************************************//
		700:
			SC_P3_ZdvizkaPredLeakTestB.StepName:='700 - Manualny Rezim';
			SC_P3_ZdvizkaPredLeakTestB.IdleTime.PT:= T#8s;
			SC_P3_ZdvizkaPredLeakTestB.AlarmTime.PT:= T#5s;

	END_CASE

	END_PROGRAM

PROGRAM _EXIT
						(* Insert code here *)

						END_PROGRAM
```

#### Variables.var - Local variables
```iecst
VAR
	SC_OvlZdvizky : SequenceControlTyp;
	Zdvizku_VYSUN : BOOL;
	Zdvizku_ZASUN : BOOL;
	Zdvizku_VYSTRED : BOOL := FALSE;
END_VAR
```

#### OvlZdvizky.st
```iecst
ACTION OvlZdvizky:

	//Volanie funkcie SequenceControl//
	SequenceControl(SC:= SC_OvlZdvizky);

	CASE SC_OvlZdvizky.Step OF

		0:
			SC_OvlZdvizky.StepName:= '0 - Nulovanie';
			Zdvizku_VYSUN:= FALSE;
			Zdvizku_ZASUN:= FALSE;
			Zdvizku_VYSTRED:= FALSE;

			IF SC_P3_ZdvizkaPredLeakTestB.Step <> 0 THEN
				SC_OvlZdvizky.ResetStep:= TRUE;
				SC_OvlZdvizky.Step:= 1;
			END_IF

		1:
			SC_OvlZdvizky.StepName:= '1 - Rozhodnutie o cinnosti';
			IF Zdvizku_VYSUN THEN
				SC_OvlZdvizky.Step:= 10;
			ELSIF Zdvizku_ZASUN THEN
				SC_OvlZdvizky.Step:= 20;
			ELSIF Zdvizku_VYSTRED THEN
				SC_OvlZdvizky.Step:= 30;
			END_IF

		10:
			SC_OvlZdvizky.StepName:= '10 - Vysunutie zdvizky hore';
			SC_OvlZdvizky.IdleTime.PT:= T#3s;
			SC_OvlZdvizky.AlarmTime.PT:= T#6s;

			IF P3_ZdvizkaPredLeakTestB.Automat THEN
				SC_OvlZdvizky.AlarmTime.IN:= TRUE;
			ELSE
				SC_OvlZdvizky.IdleTime.IN:= TRUE;
			END_IF

			IF NOT SC_OvlZdvizky.Switch1 THEN
				P3_ZdvizkaPredLeakTestB.OUT.Zdvizku_ZASUN:= FALSE;
				P3_ZdvizkaPredLeakTestB.OUT.Zdvizku_VYSUN:= TRUE;
				SC_OvlZdvizky.Switch1:= TRUE;
			END_IF

			IF P3_ZdvizkaPredLeakTestB.IN.Zdvizka_HornaPoloha OR SC_OvlZdvizky.IdleTime.Q THEN
				SC_OvlZdvizky.ResetStep:= TRUE;
				SC_OvlZdvizky.Step:= 0;
			ELSIF SC_OvlZdvizky.AlarmTime.Q THEN
				P34_Alarmy[371]:= TRUE;
				P3_Pracovisko.STAV.Porucha_ST4:= TRUE;
			END_IF

		20:
			SC_OvlZdvizky.StepName:= '20 - Zasunutie zdvizky dole';
			SC_OvlZdvizky.IdleTime.PT:= T#3s;
			SC_OvlZdvizky.AlarmTime.PT:= T#6s;

			IF P3_ZdvizkaPredLeakTestB.Automat THEN
				SC_OvlZdvizky.AlarmTime.IN:= TRUE;
			ELSE
				SC_OvlZdvizky.IdleTime.IN:= TRUE;
			END_IF

			IF NOT SC_OvlZdvizky.Switch1 THEN
				P3_ZdvizkaPredLeakTestB.OUT.Zdvizku_VYSUN:= FALSE;
				P3_ZdvizkaPredLeakTestB.OUT.Zdvizku_ZASUN:= TRUE;
				SC_OvlZdvizky.Switch1:= TRUE;
			END_IF

			IF P3_ZdvizkaPredLeakTestB.IN.Zdvizka_SpodnaPoloha OR SC_OvlZdvizky.IdleTime.Q THEN
				SC_OvlZdvizky.ResetStep:= TRUE;
				SC_OvlZdvizky.Step:= 0;
			ELSIF SC_OvlZdvizky.AlarmTime.Q THEN
				P34_Alarmy[372]:= TRUE;
				P3_Pracovisko.STAV.Porucha_ST4:= TRUE;
			END_IF

		30:
			SC_OvlZdvizky.StepName:= '30 - Presun zdvizky do strednej polohy';
			SC_OvlZdvizky.IdleTime.PT:= T#3s;
			SC_OvlZdvizky.AlarmTime.PT:= T#6s;

			IF P3_ZdvizkaPredLeakTestB.Automat THEN
				SC_OvlZdvizky.AlarmTime.IN:= TRUE;
			ELSE
				SC_OvlZdvizky.IdleTime.IN:= TRUE;
			END_IF

			IF NOT SC_OvlZdvizky.Switch1 THEN
				P3_ZdvizkaPredLeakTestB.OUT.Zdvizku_VYSUN:= FALSE;
				P3_ZdvizkaPredLeakTestB.OUT.Zdvizku_ZASUN:= FALSE;
				SC_OvlZdvizky.Switch1:= TRUE;
			END_IF

			IF P3_ZdvizkaPredLeakTestB.IN.Zdvizka_StrednaPoloha OR SC_OvlZdvizky.IdleTime.Q THEN
				SC_OvlZdvizky.ResetStep:= TRUE;
				SC_OvlZdvizky.Step:= 0;
			ELSIF SC_OvlZdvizky.AlarmTime.Q THEN
				P34_Alarmy[373]:= TRUE;
				P3_Pracovisko.STAV.Porucha_ST4:= TRUE;
			END_IF

	END_CASE

END_ACTION
```

### Program Logical/Program/Pracovisko_3/P3_LeakageTestA (IEC)

#### Main.st - Init, cyclic, exit code
```iecst
PROGRAM _INIT
	(* Insert code here *)

END_PROGRAM

PROGRAM _CYCLIC

	//Volanie funkcie SequenceControl//
	SequenceControl(SC:= SC_P3_LeakageTestA);

	//Volanie podprogramov//
	OvlCentrovacky;
	OvlHornehoPritlaku;
	IOLinkKomunikacia;
	COM_Tester;

	//Reset sekcie //
	IF P3_LeakageTestA.Reset THEN
		SC_P3_LeakageTestA.Step:= 0;
		P3_LeakageTestA.Reset:= FALSE;
	ELSIF NOT Safety.STAV.Linka_ZonaCS_AKTIVNA THEN
		SC_P3_LeakageTestA.Step:= 0;
	END_IF

	CASE SC_P3_LeakageTestA.Step OF

		0:
			SC_P3_LeakageTestA.StepName:='0 - Nulovanie';
			SC_OvlCentrovacky.Step:= 0;
			SC_OvlHornehoPritlaku.Step:= 0;
			P3_LeakageTestA.Automat:= FALSE;
			P3_LeakageTestA.KoniecCyklu:= FALSE;
			P3_LeakageTestA.Manual:= FALSE;
			P3_LeakageTestA.STAV.PoINIT:= FALSE;
			P3_LeakageTestA.OUT.ZasunStoper:= FALSE;
			P3_LeakageTestA.OUT.Kopito_VYSUN:= FALSE;
			P3_LeakageTestA.OUT.Kopito_ZASUN:= TRUE;
			P3_LeakageTestA.RFID_hlava.PrecitajChipRFID:= FALSE;
			P3_LeakageTestA.CMD.RR_TestovaciaSekvencia_START:= FALSE;
			P3_LeakageTestA.CMD.RR_VysunSpodneKopito:= FALSE;
			P3_LeakageTestA.CMD.RR_HornyPritlak_VYSUN:= FALSE;
			P3_LeakageTestA.CMD.RR_HornyPritlak_ZASUN:= FALSE;
			P3_LeakageTestA.STAV.RR_TestovaciaSekvencia_BUSY:= FALSE;
			TRCB_P3_LeakageTestA_ST8A.CMD.VyziadajStavPaletky_TYP1:= FALSE;
			TRCB_P3_LeakageTestA_ST8A.CMD.PriradQRkodFiltra_TYP3:= FALSE;
			TRCB_P3_LeakageTestA_ST8A.CMD.OdosliStavPaletky_TYP2:= FALSE;
			TRCB_P3_LeakageTestA_ST8A.CMD.VyziadajStavPanatrace_TYP4:= FALSE;
			AteqLeakageTester_A.CitajParametreTestera:= FALSE;
			AteqLeakageTester_A.START_Testovania:= FALSE;
			P34_Vizu.ZobrazHL1_ST8:= FALSE;
			P34_Vizu.ZobrazHL3_ST8:= FALSE;
			TRCB_P3_LeakTestA_OpatovnyDopyt:= FALSE;
			TRCB_P3_LeakTestA_PaletkaNG:= FALSE;
			PocetDopytovNaServer:= 0;
			PocetOpakovaniTestu:= 0;
			OpakovanyTest:= FALSE;
			TestovaciKus:= FALSE;
			P3_LeakageTestA_Taktime.IN.START_MeraniaCasu:= FALSE;
			P3_LeakageTestA_Taktime.IN.START_MeraniaStratovehoCasu:= FALSE;

			P3_ZdvizkaPredLeakTestA.STAV.PrebiehaVyvezeniePaletkyNaTratA:= FALSE;
			P3_LeakageTestA.STAV.PrebiehaVyvezeniePaletky:= FALSE;

			IF Safety.STAV.Linka_ZonaCS_AKTIVNA AND
				Safety.STAV.P3_ZonaBunky_AKTIVNA AND
				P3_Pracovisko.STAV.HardwareBunky_OK AND
				NOT P3_Pracovisko.STAV.Porucha_ST1 AND
				NOT P3_Pracovisko.STAV.Porucha_ST2 AND
				NOT P3_Pracovisko.STAV.Porucha_ST3 AND
				NOT P3_Pracovisko.STAV.Porucha_ST4 AND
				NOT P3_Pracovisko.STAV.Porucha_ST5 AND
				NOT P3_Pracovisko.STAV.Porucha_ST6 AND
				NOT P3_Pracovisko.STAV.Porucha_ST7 AND
				NOT P3_Pracovisko.STAV.Porucha_ST8 THEN
				SC_P3_LeakageTestA.ResetStep:= TRUE;
				SC_P3_LeakageTestA.Step:= 1;
			END_IF

		1:
			SC_P3_LeakageTestA.StepName:='1 - Cakam na spustenie vyroby';
			P3_LeakageTestA.KoniecCyklu:= FALSE;
			IF P3_LeakageTestA.Automat THEN
				SC_P3_LeakageTestA.Step:= 2;
			ELSIF P3_LeakageTestA.Manual THEN
				SC_P3_LeakageTestA.Step:= 700;
			END_IF

			//********************************************************Inicializácia****************************************************************************//

		2:
			SC_P3_LeakageTestA.StepName:='2 - Inicializacia - cakam na spustenie inicializacie';
			SC_P3_LeakageTestA.IdleTime.PT:= T#500ms;
			SC_P3_LeakageTestA.AlarmTime.PT:= T#5s;
			SC_P3_LeakageTestA.IdleTime.IN:= TRUE;

			IF SC_P3_LeakageTestA.IdleTime.Q THEN
				SC_P3_LeakageTestA.ResetStep:= TRUE;
				SC_P3_LeakageTestA.Step:= 5;
			END_IF

		5:
			SC_P3_LeakageTestA.StepName:='5 - Inicializacia - zasunutie horneho pritlaku';
			SC_P3_LeakageTestA.IdleTime.PT:= T#2s;
			SC_P3_LeakageTestA.AlarmTime.PT:= T#5s;

			IF NOT SC_P3_LeakageTestA.Switch1 THEN
				HornyPritlak_ZASUN:= TRUE;
				SC_P3_LeakageTestA.Switch1:= TRUE;
			END_IF

			IF P3_LeakageTestA.IN.HornyPritlak_ZASUNUTY THEN
				SC_P3_LeakageTestA.ResetStep:= TRUE;
				SC_P3_LeakageTestA.Step:= 8;
			END_IF

		8:
			SC_P3_LeakageTestA.StepName:='8 - Inicializacia - zasunutie centrovacky';
			SC_P3_LeakageTestA.IdleTime.PT:= T#4s;
			SC_P3_LeakageTestA.AlarmTime.PT:= T#5s;

			IF NOT SC_P3_LeakageTestA.Switch1 THEN
				Centrovacku_ZASUN:= TRUE;
				SC_P3_LeakageTestA.Switch1:= TRUE;
			END_IF

			IF P3_LeakageTestA.IN.Centrovanie_ZASUNUTE THEN
				SC_P3_LeakageTestA.ResetStep:= TRUE;
				SC_P3_LeakageTestA.Step:= 10;
			END_IF

		10:
			SC_P3_LeakageTestA.StepName:='10 - Inicializacia - kontrola typu zalozeneho kopita';
			SC_P3_LeakageTestA.IdleTime.PT:= T#4s;
			SC_P3_LeakageTestA.AlarmTime.PT:= T#5s;

			IF Linka.PAR.ZvolenyModel = '4F' AND P3_LeakageTestA.IN.PritomnostKopita AND P3_LeakageTestA.IN.Tester_TypKonektoru_4F THEN
				SC_P3_LeakageTestA.ResetStep:= TRUE;
				SC_P3_LeakageTestA.Step:= 13;
			ELSIF Linka.PAR.ZvolenyModel = '5F' AND P3_LeakageTestA.IN.PritomnostKopita AND P3_LeakageTestA.IN.Tester_TypKonektoru_5F_5H THEN
				SC_P3_LeakageTestA.ResetStep:= TRUE;
				SC_P3_LeakageTestA.Step:= 13;
			ELSIF Linka.PAR.ZvolenyModel = '5H' AND P3_LeakageTestA.IN.PritomnostKopita AND P3_LeakageTestA.IN.Tester_TypKonektoru_5F_5H THEN
				SC_P3_LeakageTestA.ResetStep:= TRUE;
				SC_P3_LeakageTestA.Step:= 13;
			ELSE
				P34_Alarmy[314]:= TRUE;
				P3_Pracovisko.STAV.Porucha_ST5:= TRUE;
			END_IF

		13:
			SC_P3_LeakageTestA.StepName:='13 - Inicializacia - hladanie paletky';
			SC_P3_LeakageTestA.IdleTime.PT:= T#5s;
			SC_P3_LeakageTestA.AlarmTime.PT:= T#5s;

			SC_P3_LeakageTestA.IdleTime.IN:= P3_Dopravniky.STAV.PoINIT;

			IF P3_LeakageTestA.CMD.RR_TestovaciaSekvencia_START THEN
				SC_P3_LeakageTestA.ResetStep:= TRUE;
				SC_P3_LeakageTestA.Step:= 120;
			ELSIF P3_LeakageTestA.RFID_hlava.PritomnostPaletky THEN
				SC_P3_LeakageTestA.ResetStep:= TRUE;
				SC_P3_LeakageTestA.Step:= 20;
			ELSIF SC_P3_LeakageTestA.IdleTime.Q THEN
				P3_LeakageTestA.STAV.PoINIT:= TRUE;
				SC_P3_LeakageTestA.ResetStep:= TRUE;
				SC_P3_LeakageTestA.Step:= 100;
			END_IF

		20:
			SC_P3_LeakageTestA.StepName:='20 - Inicializacia - precitanie cisla paletky';
			SC_P3_LeakageTestA.IdleTime.PT:= T#200ms;
			SC_P3_LeakageTestA.AlarmTime.PT:= T#5s;

			SC_P3_LeakageTestA.IdleTime.IN:= P3_LeakageTestA.RFID_hlava.PritomnostPaletky;

			IF SC_P3_LeakageTestA.IdleTime.Q AND NOT SC_P3_LeakageTestA.Switch1 THEN
				P3_LeakageTestA.RFID_hlava.PrecitajChipRFID:= TRUE;
				i:= 0;
				SC_P3_LeakageTestA.Switch1:= TRUE;
			END_IF

			IF P3_LeakageTestA.RFID_hlava.Stav_CitanieZapis_OK AND P3_LeakageTestA.RFID_hlava.PrecitaneCisloPaletky <> 0 THEN
				i:= P3_LeakageTestA.RFID_hlava.PrecitaneCisloPaletky;
				P3_LeakageTestA.PAR.CisloPaletky:= P3_LeakageTestA.RFID_hlava.PrecitaneCisloPaletky;
				P3_LeakageTestA.RFID_hlava.PrecitajChipRFID:= FALSE;
				SC_P3_LeakageTestA.ResetStep:= TRUE;
				SC_P3_LeakageTestA.Step:= 23;
			END_IF

		23:
			SC_P3_LeakageTestA.StepName:='23 - Inicializacia - priradenie indexu paletky na zaklade precitanej hodnoty';
			SC_P3_LeakageTestA.IdleTime.PT:= T#200ms;
			SC_P3_LeakageTestA.AlarmTime.PT:= T#5s;

			IF i<> 0 THEN
				P3_LeakageTestA.PAR.CisloPaletky_STRING:= USINT_TO_STRING(i);
				Paletka[i].PAR.CisloPaletky:= USINT_TO_STRING(i);
				SC_P3_LeakageTestA.ResetStep:= TRUE;
				SC_P3_LeakageTestA.Step:= 30;
			ELSE
				P34_Alarmy[310]:= TRUE;
				P3_Pracovisko.STAV.Porucha_ST5:= TRUE;
			END_IF

		30:
			SC_P3_LeakageTestA.StepName:='30 - Inicializacia - kontrola stavu paletky';
			SC_P3_LeakageTestA.IdleTime.PT:= T#200ms;
			SC_P3_LeakageTestA.AlarmTime.PT:= T#5s;

			IF Paletka[i].STAV.StavPaletky = '' THEN
				Paletka[i].STAV.StavPaletky:= 'NG';
				SC_P3_LeakageTestA.ResetStep:= TRUE;
				SC_P3_LeakageTestA.Step:= 560;
			ELSIF Paletka[i].STAV.StavPaletky = 'PRECH' THEN
				P3_LeakageTestA.STAV.PoINIT:= TRUE;
				SC_P3_LeakageTestA.ResetStep:= TRUE;
				SC_P3_LeakageTestA.Step:= 560;
			ELSIF Paletka[i].STAV.StavPaletky = 'TEST' AND Paletka[i].STAV.CisloTestovacejStanice = 'ST_8A,8B' THEN
				IF P3_LeakageTestA.STAV.Tester_ON THEN
					TestovaciKus:= TRUE;
					P3_LeakageTestA.STAV.PoINIT:= TRUE;
					SC_P3_LeakageTestA.ResetStep:= TRUE;
					SC_P3_LeakageTestA.Step:= 110;
				ELSE
					P3_LeakageTestA.STAV.PoINIT:= TRUE;
					SC_P3_LeakageTestA.ResetStep:= TRUE;
					SC_P3_LeakageTestA.Step:= 560;
				END_IF
			ELSIF Paletka[i].STAV.StavPaletky = 'TEST' AND Paletka[i].STAV.CisloTestovacejStanice <> 'ST_8A,8B' THEN
				P3_LeakageTestA.STAV.PoINIT:= TRUE;
				SC_P3_LeakageTestA.ResetStep:= TRUE;
				SC_P3_LeakageTestA.Step:= 560;
			ELSIF Paletka[i].STAV.StavPaletky = 'REV' AND Paletka[i].STAV.CisloRevorkovejStanice = 'ST_8A,8B' THEN
				IF P3_LeakageTestA.STAV.Tester_ON THEN
					Paletka[i].STAV.StavPaletky:= 'OK';
					P3_LeakageTestA.STAV.PoINIT:= TRUE;
					SC_P3_LeakageTestA.ResetStep:= TRUE;
					SC_P3_LeakageTestA.Step:= 110;
				ELSE
					P3_LeakageTestA.STAV.PoINIT:= TRUE;
					SC_P3_LeakageTestA.ResetStep:= TRUE;
					SC_P3_LeakageTestA.Step:= 560;
				END_IF
			ELSIF Paletka[i].STAV.StavPaletky = 'REV' AND Paletka[i].STAV.CisloRevorkovejStanice <> 'ST_8A,8B' THEN
				P3_LeakageTestA.STAV.PoINIT:= TRUE;
				SC_P3_LeakageTestA.ResetStep:= TRUE;
				SC_P3_LeakageTestA.Step:= 560;
			ELSIF Paletka[i].STAV.StavPaletky = 'OK' THEN
				IF P3_LeakageTestA.STAV.Tester_ON THEN
					SC_P3_LeakageTestA.ResetStep:= TRUE;
					SC_P3_LeakageTestA.Step:= 33;
				ELSE
					P3_LeakageTestA.STAV.PoINIT:= TRUE;
					SC_P3_LeakageTestA.ResetStep:= TRUE;
					SC_P3_LeakageTestA.Step:= 560;
				END_IF
			ELSIF Paletka[i].STAV.StavPaletky = 'NG' THEN
				P3_LeakageTestA.STAV.PoINIT:= TRUE;
				SC_P3_LeakageTestA.ResetStep:= TRUE;
				SC_P3_LeakageTestA.Step:= 560;
			END_IF

		33:
			SC_P3_LeakageTestA.StepName:='33 - Inicializacia - kontrola uzavretia komunikacie';
			SC_P3_LeakageTestA.IdleTime.PT:= T#200ms;
			SC_P3_LeakageTestA.AlarmTime.PT:= T#5s;

			IF Paletka[i].STAV.Komunikacia_DONE THEN
				P3_LeakageTestA.STAV.PoINIT:= TRUE;
				SC_P3_LeakageTestA.ResetStep:= TRUE;
				SC_P3_LeakageTestA.Step:= 560;
			ELSE
				P3_LeakageTestA.STAV.PoINIT:= TRUE;
				SC_P3_LeakageTestA.ResetStep:= TRUE;
				SC_P3_LeakageTestA.Step:= 100;
			END_IF

			//********************************************************Automatický režim****************************************************************************//

		100:
			SC_P3_LeakageTestA.StepName:='100 - Automaticky Rezim - cakam na príchod paletky na stoper';
			SC_P3_LeakageTestA.IdleTime.PT:= T#200ms;
			SC_P3_LeakageTestA.AlarmTime.PT:= T#5s;

			SC_P3_LeakageTestA.IdleTime.IN:= P3_LeakageTestA.RFID_hlava.PritomnostPaletky;

			IF P3_LeakageTestA.RFID_hlava.PritomnostPaletky THEN
				P3_ZdvizkaPredLeakTestA.STAV.PrebiehaVyvezeniePaletkyNaTratA:= FALSE;
			END_IF

			IF NOT SC_P3_LeakageTestA.Switch1 AND P3_LeakageTestA.RFID_hlava.PritomnostPaletky THEN
				P3_LeakageTestA_Taktime.IN.START_MeraniaCasu:= TRUE;
				P3_LeakageTestA_Taktime.IN.ZAPIS_MeraniaCasu:= TRUE;
				P3_LeakageTestA_Taktime.IN.ZAPIS_StratovyCas:= TRUE;
				Buffer_9.Hodnota:= P3_LeakageTestA_Taktime.OUT.StratoveSekundy;
				Buffer_9.ZapisHodnotu:= TRUE;
				SC_P3_LeakageTestA.Switch1:= TRUE;
			END_IF

			IF P3_LeakageTestA.KoniecCyklu THEN
				SC_P3_LeakageTestA.ResetStep:= TRUE;
				SC_P3_LeakageTestA.Step:= 0;
			ELSIF SC_P3_LeakageTestA.IdleTime.Q THEN
				SC_P3_LeakageTestA.ResetStep:= TRUE;
				SC_P3_LeakageTestA.Step:= 101;
			END_IF

		101:
			SC_P3_LeakageTestA.StepName:='101 - Automaticky Rezim - precitanie cisla paletky';
			SC_P3_LeakageTestA.IdleTime.PT:= T#200ms;
			SC_P3_LeakageTestA.AlarmTime.PT:= T#5s;
			SC_P3_LeakageTestA.IdleTime.IN:= TRUE;

			IF NOT SC_P3_LeakageTestA.Switch1 THEN
				P3_LeakageTestA.RFID_hlava.PrecitajChipRFID:= TRUE;
				i:= 0;
				SC_P3_LeakageTestA.Switch1:= TRUE;
			END_IF

			IF P3_LeakageTestA.RFID_hlava.Stav_CitanieZapis_OK AND P3_LeakageTestA.RFID_hlava.PrecitaneCisloPaletky <> 0 THEN
				i:= P3_LeakageTestA.RFID_hlava.PrecitaneCisloPaletky;
				P3_LeakageTestA.PAR.CisloPaletky:= P3_LeakageTestA.RFID_hlava.PrecitaneCisloPaletky;
				P3_LeakageTestA.RFID_hlava.PrecitajChipRFID:= FALSE;
				SC_P3_LeakageTestA.ResetStep:= TRUE;
				SC_P3_LeakageTestA.Step:= 102;
			END_IF

		102:
			SC_P3_LeakageTestA.StepName:='102 - Automaticky Rezim - priradenie indexu paletky na zaklade precitanej hodnoty';
			SC_P3_LeakageTestA.IdleTime.PT:= T#200ms;
			SC_P3_LeakageTestA.AlarmTime.PT:= T#5s;

			IF i<> 0 THEN
				P3_LeakageTestA.PAR.CisloPaletky_STRING:= USINT_TO_STRING(i);
				Paletka[i].PAR.CisloPaletky:= USINT_TO_STRING(i);
				SC_P3_LeakageTestA.ResetStep:= TRUE;
				SC_P3_LeakageTestA.Step:= 103;
			ELSE
				P34_Alarmy[310]:= TRUE;
				P3_Pracovisko.STAV.Porucha_ST5:= TRUE;
			END_IF

		103:
			SC_P3_LeakageTestA.StepName:='103 - Automaticky Rezim - kontrola stavu paletky';
			SC_P3_LeakageTestA.IdleTime.PT:= T#200ms;
			SC_P3_LeakageTestA.AlarmTime.PT:= T#5s;

			IF Paletka[i].STAV.StavPaletky = '' THEN
				Paletka[i].STAV.StavPaletky:= 'NG';
				SC_P3_LeakageTestA.ResetStep:= TRUE;
				SC_P3_LeakageTestA.Step:= 560;
			ELSIF Paletka[i].STAV.StavPaletky = 'PRECH' THEN
				SC_P3_LeakageTestA.ResetStep:= TRUE;
				SC_P3_LeakageTestA.Step:= 560;
			ELSIF Paletka[i].STAV.StavPaletky = 'TEST' AND Paletka[i].STAV.CisloTestovacejStanice = 'ST_8A,8B' THEN
				IF P3_LeakageTestA.STAV.Tester_ON THEN
					TestovaciKus:= TRUE;
					SC_P3_LeakageTestA.ResetStep:= TRUE;
					SC_P3_LeakageTestA.Step:= 110;
				ELSE
					SC_P3_LeakageTestA.ResetStep:= TRUE;
					SC_P3_LeakageTestA.Step:= 560;
				END_IF
			ELSIF Paletka[i].STAV.StavPaletky = 'TEST' AND Paletka[i].STAV.CisloTestovacejStanice <> 'ST_8A,8B' THEN
				SC_P3_LeakageTestA.ResetStep:= TRUE;
				SC_P3_LeakageTestA.Step:= 560;
			ELSIF Paletka[i].STAV.StavPaletky = 'REV' AND Paletka[i].STAV.CisloRevorkovejStanice = 'ST_8A,8B' THEN
				IF P3_LeakageTestA.STAV.Tester_ON THEN
					Paletka[i].STAV.StavPaletky:= 'OK';
					SC_P3_LeakageTestA.ResetStep:= TRUE;
					SC_P3_LeakageTestA.Step:= 110;
				ELSE
					SC_P3_LeakageTestA.ResetStep:= TRUE;
					SC_P3_LeakageTestA.Step:= 560;
				END_IF
			ELSIF Paletka[i].STAV.StavPaletky = 'REV' AND Paletka[i].STAV.CisloRevorkovejStanice <> 'ST_8A,8B' THEN
				SC_P3_LeakageTestA.ResetStep:= TRUE;
				SC_P3_LeakageTestA.Step:= 560;
			ELSIF Paletka[i].STAV.StavPaletky = 'OK' THEN
				IF P3_LeakageTestA.STAV.Tester_ON THEN
					SC_P3_LeakageTestA.ResetStep:= TRUE;
					SC_P3_LeakageTestA.Step:= 110;
				ELSE
					SC_P3_LeakageTestA.ResetStep:= TRUE;
					SC_P3_LeakageTestA.Step:= 560;
				END_IF
			ELSIF Paletka[i].STAV.StavPaletky = 'NG' THEN
				SC_P3_LeakageTestA.ResetStep:= TRUE;
				SC_P3_LeakageTestA.Step:= 560;
			END_IF

		110:
			SC_P3_LeakageTestA.StepName:='110 - Automaticky Rezim - vyziadanie stavu komunikacie zo serverom';
			SC_P3_LeakageTestA.IdleTime.PT:= T#200ms;
			SC_P3_LeakageTestA.AlarmTime.PT:= T#10s;

			IF Linka.KOM_Panatrace_OFF THEN
				SC_P3_LeakageTestA.ResetStep:= TRUE;
				SC_P3_LeakageTestA.Step:= 120;
			ELSIF NOT SC_P3_LeakageTestA.Switch1 AND TRCB_P3_LeakageTestA_ST8A.STATUS.KOM_READY THEN
				TRCB_P3_LeakageTestA_ST8A.CMD.VyziadajStavPanatrace_TYP4:= TRUE;
				Centrovacku_VYSUN:= TRUE;
				P3_LeakageTestA_Taktime.IN.START_MeraniaStratovehoCasu:= TRUE;
				SC_P3_LeakageTestA.Switch1:= TRUE;
			END_IF

			IF TRCB_P3_LeakageTestA_ST8A.STATUS.KomunikaciaUkoncena THEN
				TRCB_P3_LeakageTestA_ST8A.CMD.VyziadajStavPanatrace_TYP4:= FALSE;
				P3_LeakageTestA_Taktime.IN.START_MeraniaStratovehoCasu:= FALSE;
				SC_P3_LeakageTestA.ResetStep:= TRUE;
				SC_P3_LeakageTestA.Step:= 111;
			ELSIF TRCB_P3_LeakageTestA_ST8A.STATUS.KomunikaciaError THEN
				TRCB_P3_LeakageTestA_ST8A.CMD.VyziadajStavPanatrace_TYP4:= FALSE;
				P3_LeakageTestA_Taktime.IN.START_MeraniaStratovehoCasu:= FALSE;
				SC_P3_LeakageTestA.ResetStep:= TRUE;
				SC_P3_LeakageTestA.Step:= 112;
			END_IF

		111:
			SC_P3_LeakageTestA.StepName:='111 - Automaticky Rezim - kontrola odpovede servera';
			SC_P3_LeakageTestA.IdleTime.PT:= T#200ms;
			SC_P3_LeakageTestA.AlarmTime.PT:= T#5s;

			IF NOT TRCB_P3_LeakageTestA_ST8A.STATUS.KomunikaciaUkoncena THEN
				IF TRCB_P3_LeakageTestA_ST8A.OUTPUTS.DruhCinnostiNaPaletke = '0;Generating' THEN
					SC_P3_LeakageTestA.ResetStep:= TRUE;
					SC_P3_LeakageTestA.Step:= 112;
				ELSIF TRCB_P3_LeakageTestA_ST8A.OUTPUTS.DruhCinnostiNaPaletke = '1;Request' THEN
					SC_P3_LeakageTestA.ResetStep:= TRUE;
					SC_P3_LeakageTestA.Step:= 115;
				ELSIF TRCB_P3_LeakageTestA_ST8A.OUTPUTS.DruhCinnostiNaPaletke = '2;Report' THEN
					SC_P3_LeakageTestA.ResetStep:= TRUE;
					SC_P3_LeakageTestA.Step:= 120;
				ELSIF TRCB_P3_LeakageTestA_ST8A.OUTPUTS.DruhCinnostiNaPaletke = '3;Wedding' THEN
					SC_P3_LeakageTestA.ResetStep:= TRUE;
					SC_P3_LeakageTestA.Step:= 112;
				ELSIF TRCB_P3_LeakageTestA_ST8A.OUTPUTS.DruhCinnostiNaPaletke = '4;Status' THEN
					SC_P3_LeakageTestA.ResetStep:= TRUE;
					SC_P3_LeakageTestA.Step:= 112;
				ELSIF TRCB_P3_LeakageTestA_ST8A.OUTPUTS.DruhCinnostiNaPaletke = '5;' THEN
					SC_P3_LeakageTestA.ResetStep:= TRUE;
					SC_P3_LeakageTestA.Step:= 112;
				ELSE
					SC_P3_LeakageTestA.ResetStep:= TRUE;
					SC_P3_LeakageTestA.Step:= 112;
				END_IF
			END_IF

		112:
			SC_P3_LeakageTestA.StepName:='112 - Automaticky Rezim - rozhodnutie obsluhy po chybe komunikacie s Panatrace';
			SC_P3_LeakageTestA.IdleTime.PT:= T#200ms;
			SC_P3_LeakageTestA.AlarmTime.PT:= T#5s;

			P34_Vizu.ZobrazHL3_ST8:= TRUE;

			IF TRCB_P3_LeakTestA_OpatovnyDopyt THEN
				TRCB_P3_LeakTestA_OpatovnyDopyt:= FALSE;
				P34_Vizu.ZobrazHL3_ST8:= FALSE;
				SC_P3_LeakageTestA.ResetStep:= TRUE;
				SC_P3_LeakageTestA.Step:= 110;
			ELSIF TRCB_P3_LeakTestA_PaletkaNG THEN
				TRCB_P3_LeakTestA_PaletkaNG:= FALSE;
				P34_Vizu.ZobrazHL3_ST8:= FALSE;
				Paletka[i].STAV.StavPaletky := 'NG';
				SC_P3_LeakageTestA.ResetStep:= TRUE;
				SC_P3_LeakageTestA.Step:= 118;
			END_IF

		115:
			SC_P3_LeakageTestA.StepName:='115 - Automaticky Rezim - vyziadanie stavu paletky zo servera, zacentrovanie paletky';
			SC_P3_LeakageTestA.IdleTime.PT:= T#200ms;
			SC_P3_LeakageTestA.AlarmTime.PT:= T#5s;
			SC_P3_LeakageTestA.IdleTime.IN:= TRUE;

			IF NOT SC_P3_LeakageTestA.Switch1 AND TRCB_P3_LeakageTestA_ST8A.STATUS.KOM_READY THEN
				TRCB_P3_LeakageTestA_ST8A.CMD.VyziadajStavPaletky_TYP1:= TRUE;
				P3_LeakageTestA_Taktime.IN.START_MeraniaStratovehoCasu:= TRUE;
				SC_P3_LeakageTestA.Switch1:= TRUE;
			END_IF

			IF TRCB_P3_LeakageTestA_ST8A.STATUS.KomunikaciaUkoncena THEN
				TRCB_P3_LeakageTestA_ST8A.CMD.VyziadajStavPaletky_TYP1:= FALSE;
				P3_LeakageTestA_Taktime.IN.START_MeraniaStratovehoCasu:= FALSE;
				SC_P3_LeakageTestA.ResetStep:= TRUE;
				SC_P3_LeakageTestA.Step:= 116;
			ELSIF TRCB_P3_LeakageTestA_ST8A.STATUS.KomunikaciaError THEN
				TRCB_P3_LeakageTestA_ST8A.CMD.VyziadajStavPaletky_TYP1:= FALSE;
				P3_LeakageTestA_Taktime.IN.START_MeraniaStratovehoCasu:= FALSE;
				SC_P3_LeakageTestA.ResetStep:= TRUE;
				SC_P3_LeakageTestA.Step:= 112;
			END_IF

		116:
			SC_P3_LeakageTestA.StepName:='116 - Automaticky Rezim - kontrola odpovede servera';
			SC_P3_LeakageTestA.IdleTime.PT:= T#200ms;
			SC_P3_LeakageTestA.AlarmTime.PT:= T#5s;

			IF NOT TRCB_P3_LeakageTestA_ST8A.STATUS.KomunikaciaUkoncena AND P3_LeakageTestA.IN.Centrovanie_VYSUNUTE THEN
				IF TRCB_P3_LeakageTestA_ST8A.OUTPUTS.PovolenieCinnostiNaPaletke = 'OK' THEN
					IF TRCB_P3_LeakageTestA_ST8A.OUTPUTS.DruhCinnostiNaPaletke  = 'PRD;ST8A' THEN
						SC_P3_LeakageTestA.ResetStep:= TRUE;
						SC_P3_LeakageTestA.Step:= 120;
					ELSIF TRCB_P3_LeakageTestA_ST8A.OUTPUTS.DruhCinnostiNaPaletke  = 'SMP;ST8A,ST8B' THEN
						SC_P3_LeakageTestA.ResetStep:= TRUE;
						SC_P3_LeakageTestA.Step:= 120;
					ELSIF TRCB_P3_LeakageTestA_ST8A.OUTPUTS.DruhCinnostiNaPaletke  = 'PRD;ST8A,ST8B' THEN
						SC_P3_LeakageTestA.ResetStep:= TRUE;
						SC_P3_LeakageTestA.Step:= 120;
					END_IF
				ELSIF TRCB_P3_LeakageTestA_ST8A.OUTPUTS.PovolenieCinnostiNaPaletke = 'NG' THEN
					SC_P3_LeakageTestA.ResetStep:= TRUE;
					SC_P3_LeakageTestA.Step:= 117;
				END_IF
			END_IF

		117:
			SC_P3_LeakageTestA.StepName:='115 - Automaticky Rezim - rozhodnutie obsluhy po odpovedi panatrace NG';
			SC_P3_LeakageTestA.IdleTime.PT:= T#200ms;
			SC_P3_LeakageTestA.AlarmTime.PT:= T#5s;

			P34_Vizu.ZobrazHL1_ST8:= TRUE;

			IF TRCB_P3_LeakTestA_OpatovnyDopyt THEN
				TRCB_P3_LeakTestA_OpatovnyDopyt:= FALSE;
				P34_Vizu.ZobrazHL1_ST8:= FALSE;
				SC_P3_LeakageTestA.ResetStep:= TRUE;
				SC_P3_LeakageTestA.Step:= 110;
			ELSIF TRCB_P3_LeakTestA_PaletkaNG THEN
				TRCB_P3_LeakTestA_PaletkaNG:= FALSE;
				P34_Vizu.ZobrazHL1_ST8:= FALSE;
				Paletka[i].STAV.StavPaletky := 'NG';
				SC_P3_LeakageTestA.ResetStep:= TRUE;
				SC_P3_LeakageTestA.Step:= 118;
			END_IF

		118:
			SC_P3_LeakageTestA.StepName:='118 - Automaticky Rezim - odcentrovanie paletky po odpovedi servera NG';
			SC_P3_LeakageTestA.IdleTime.PT:= T#200ms;
			SC_P3_LeakageTestA.AlarmTime.PT:= T#5s;

			IF NOT SC_P3_LeakageTestA.Switch1 THEN
				Centrovacku_ZASUN:= TRUE;
				SC_P3_LeakageTestA.Switch1:= TRUE;
			END_IF

			IF P3_LeakageTestA.IN.Centrovanie_ZASUNUTE THEN
				SC_P3_LeakageTestA.ResetStep:= TRUE;
				SC_P3_LeakageTestA.Step:= 560;
			END_IF

			//Zatvorenie Leakage testera//

		120:
			SC_P3_LeakageTestA.StepName:='120 - Automaticky Rezim - zacentrovanie paletky ';
			SC_P3_LeakageTestA.IdleTime.PT:= T#200ms;
			SC_P3_LeakageTestA.AlarmTime.PT:= T#5s;

			IF NOT SC_P3_LeakageTestA.Switch1 THEN
				Centrovacku_VYSUN:= TRUE;
				SC_P3_LeakageTestA.Switch1:= TRUE;
			END_IF

			IF P3_LeakageTestA.IN.Centrovanie_VYSUNUTE THEN
				SC_P3_LeakageTestA.ResetStep:= TRUE;
				SC_P3_LeakageTestA.Step:= 123;
			END_IF

		123:
			SC_P3_LeakageTestA.StepName:='123 - Automaticky Rezim - vysunutie horneho pritlaku ';
			SC_P3_LeakageTestA.IdleTime.PT:= T#3s;
			SC_P3_LeakageTestA.AlarmTime.PT:= T#5s;

			IF NOT SC_P3_LeakageTestA.Switch1 THEN
				HornyPritlak_VYSUN:= TRUE;
				SC_P3_LeakageTestA.Switch1:= TRUE;
			END_IF

			IF P3_LeakageTestA.IN.HornyPritlak_VYSUNUTY THEN
				SC_P3_LeakageTestA.ResetStep:= TRUE;
				SC_P3_LeakageTestA.Step:= 125;
			END_IF

		125:
			SC_P3_LeakageTestA.StepName:='125 - Automaticky Rezim - vysunutie spodneho kopita';
			SC_P3_LeakageTestA.IdleTime.PT:= T#1s;
			SC_P3_LeakageTestA.AlarmTime.PT:= T#5s;
			SC_P3_LeakageTestA.IdleTime.IN:= TRUE;

			IF P3_LeakageTestA.IN.PritomnostKopita AND P3_LeakageTestA.IN.Kopito_ZASUNUTE THEN
				P3_LeakageTestA.OUT.Kopito_ZASUN:= FALSE;
				P3_LeakageTestA.OUT.Kopito_VYSUN:= TRUE;
				SC_P3_LeakageTestA.ResetStep:= TRUE;
				SC_P3_LeakageTestA.Step:= 128;
			END_IF

		128:
			SC_P3_LeakageTestA.StepName:='128 - Automaticky Rezim - cakam na vysunutie kopita, zamknutie pneuzamkov';
			SC_P3_LeakageTestA.IdleTime.PT:= T#200ms;
			SC_P3_LeakageTestA.AlarmTime.PT:= T#300ms;

			SC_P3_LeakageTestA.IdleTime.IN:= NOT P3_LeakageTestA.IN.Kopito_ZASUNUTE;

			IF SC_P3_LeakageTestA.IdleTime.Q THEN
				P3_LeakageTestA.OUT.PneuZamokCentrovania_ODOMKNI:= FALSE;
				P3_LeakageTestA.OUT.PneuZamokZvonu_ODOMKNI:= FALSE;
				SC_P3_LeakageTestA.ResetStep:= TRUE;
				SC_P3_LeakageTestA.Step:= 130;
			END_IF

		130:
			SC_P3_LeakageTestA.StepName:='130 - Automaticky Rezim - spustenie testera';
			SC_P3_LeakageTestA.IdleTime.PT:= T#4s800ms;
			SC_P3_LeakageTestA.AlarmTime.PT:= T#2s;

			IF NOT SC_P3_LeakageTestA.Switch1 AND AteqLeakageTester_A.Stav_READY THEN
				AteqLeakageTester_A.START_Testovania:= TRUE;
				SC_P3_LeakageTestA.IdleTime.IN:= TRUE;
				SC_P3_LeakageTestA.Switch1:= TRUE;
			END_IF

			IF NOT AteqLeakageTester_A.Stav_READY AND AteqLeakageTester_A.Stav_START_DONE AND NOT AteqLeakageTester_A.VysledokTestovania_OK AND NOT AteqLeakageTester_A.VysledokTestovania_NG AND SC_P3_LeakageTestA.IdleTime.Q THEN
				SC_P3_LeakageTestA.ResetStep:= TRUE;
				SC_P3_LeakageTestA.Step:= 133;
			END_IF

		133:
			SC_P3_LeakageTestA.StepName:='133 - Automaticky Rezim - nacitanie parametrov testera';
			SC_P3_LeakageTestA.IdleTime.PT:= T#500ms;
			SC_P3_LeakageTestA.AlarmTime.PT:= T#5s;

			IF AteqLeakageTester_A.Stav_READY THEN
				AteqLeakageTester_A.START_Testovania:= FALSE;
				AteqLeakageTester_A.CitajParametreTestera:= TRUE;
			END_IF

			SC_P3_LeakageTestA.IdleTime.IN:= AteqLeakageTester_A.Stav_CitanieParametrov_OK;

			IF AteqLeakageTester_A.Stav_CitanieParametrov_OK AND SC_P3_LeakageTestA.IdleTime.Q THEN
				Reports.LeakageTest.CasPlnenia.StanicaA:= REAL_TO_STRING(AteqLeakageTester_A.CasPnenia);
				Reports.LeakageTest.CasStabilizacie.StanicaA:= REAL_TO_STRING(AteqLeakageTester_A.CasStabilizacie);
				Reports.LeakageTest.TlakPlnenia.StanicaA:= REAL_TO_STRING(AteqLeakageTester_A.TlakPlnenia);
				Reports.LeakageTest.ToleranciaPritlaku_MIN.StanicaA:= '';
				Reports.LeakageTest.ToleranciaPritlaku_MAX.StanicaA:= '';
				Reports.LeakageTest.TlakPritlaku.StanicaA:= REAL_TO_STRING(P3_LeakageTestA.PAR.PreratanyVyrovnavaciTlak_Bar);
				Reports.LeakageTest.TlakUniku.StanicaA:= REAL_TO_STRING(AteqLeakageTester_A.TlakUniku);
				Reports.LeakageTest.ToleranciaTlakUniku_MIN.StanicaA:= REAL_TO_STRING(AteqLeakageTester_A.Tolerancia * -1);
				Reports.LeakageTest.ToleranciaTlakUniku_MAX.StanicaA:= REAL_TO_STRING(AteqLeakageTester_A.Tolerancia);
				Reports.LeakageTest.Tolerancia.StanicaA:= REAL_TO_STRING(AteqLeakageTester_A.Tolerancia);
				AteqLeakageTester_A.CitajParametreTestera:= FALSE;
				IF P3_LeakageTestA.STAV.RR_TestovaciaSekvencia_BUSY THEN
					SC_P3_LeakageTestA.ResetStep:= TRUE;
					SC_P3_LeakageTestA.Step:= 150;
				ELSE
					SC_P3_LeakageTestA.ResetStep:= TRUE;
					SC_P3_LeakageTestA.Step:= 135;
				END_IF
			END_IF

		135:
			SC_P3_LeakageTestA.StepName:='135 - Automaticky Rezim - kontrola výsledku testu';
			SC_P3_LeakageTestA.IdleTime.PT:= T#1s;
			SC_P3_LeakageTestA.AlarmTime.PT:= T#5s;

			IF AteqLeakageTester_A.VysledokTestovania_OK THEN
				Paletka[i].STAV.LeakageTest_Ukonceny:= TRUE;
				Reports.LeakageTest.VyslednyReport.StanicaA:= 'PASS';
				Paletka[i].PAR.StavPowerCP:= 'PASS';
				IF Paletka[i].STAV.StavPaletky <> 'TEST'THEN
					Paletka[i].STAV.StavPaletky:= 'OK';
				END_IF
				PocetOpakovaniTestu:= 0;
				OpakovanyTest:= FALSE;
				SC_P3_LeakageTestA.ResetStep:= TRUE;
				SC_P3_LeakageTestA.Step:= 150;
			ELSE
				IF NOT TestovaciKus THEN
					PocetOpakovaniTestu:= PocetOpakovaniTestu + 1;
					OpakovanyTest:= TRUE;
				END_IF
				Reports.LeakageTest.VyslednyReport.StanicaA:= 'FAIL';
				Paletka[i].PAR.StavPowerCP:= 'FAIL';
				IF Paletka[i].STAV.StavPaletky <> 'TEST'THEN
					Paletka[i].STAV.StavPaletky:= 'NG';
				END_IF
				SC_P3_LeakageTestA.ResetStep:= TRUE;
				SC_P3_LeakageTestA.Step:= 150;
			END_IF

			//Otvorenie Leakage testera//

		150:
			SC_P3_LeakageTestA.StepName:='150 - Automaticky Rezim - zasunutie spodneho kopita ';
			SC_P3_LeakageTestA.IdleTime.PT:= T#200ms;
			SC_P3_LeakageTestA.AlarmTime.PT:= T#5s;

			P3_LeakageTestA.OUT.Kopito_VYSUN:= FALSE;
			P3_LeakageTestA.OUT.Kopito_ZASUN:= TRUE;

			IF P3_LeakageTestA.IN.Kopito_ZASUNUTE THEN
				SC_P3_LeakageTestA.ResetStep:= TRUE;
				SC_P3_LeakageTestA.Step:= 153;
			END_IF

		153:
			SC_P3_LeakageTestA.StepName:='153 - Automaticky Rezim - zasunutie horneho pritlaku';
			SC_P3_LeakageTestA.IdleTime.PT:= T#200ms;
			SC_P3_LeakageTestA.AlarmTime.PT:= T#5s;

			IF NOT SC_P3_LeakageTestA.Switch1 THEN
				HornyPritlak_ZASUN:= TRUE;
				Centrovacku_ZASUN:= TRUE;
				SC_P3_LeakageTestA.Switch1:= TRUE;
			END_IF

			IF P3_LeakageTestA.IN.HornyPritlak_ZASUNUTY THEN
				SC_P3_LeakageTestA.ResetStep:= TRUE;
				SC_P3_LeakageTestA.Step:= 155;
			END_IF

		155:
			SC_P3_LeakageTestA.StepName:='155 - Automaticky Rezim - odcentrovanie paletky ';
			SC_P3_LeakageTestA.IdleTime.PT:= T#200ms;
			SC_P3_LeakageTestA.AlarmTime.PT:= T#5s;

			IF NOT SC_P3_LeakageTestA.Switch1 THEN
				Centrovacku_ZASUN:= TRUE;
				SC_P3_LeakageTestA.Switch1:= TRUE;
			END_IF

			IF P3_LeakageTestA.IN.Centrovanie_ZASUNUTE THEN
				IF P3_LeakageTestA.STAV.RR_TestovaciaSekvencia_BUSY THEN
					P3_LeakageTestA.STAV.RR_TestovaciaSekvencia_BUSY:= FALSE;
					SC_P3_LeakageTestA.ResetStep:= TRUE;
					SC_P3_LeakageTestA.Step:= 700;
				ELSE
					SC_P3_LeakageTestA.ResetStep:= TRUE;
					SC_P3_LeakageTestA.Step:= 160;
				END_IF
			END_IF

		160:
			SC_P3_LeakageTestA.StepName:='160 - Automaticky Rezim - rozhodnutie o opakovani testu ';
			SC_P3_LeakageTestA.IdleTime.PT:= T#1s;
			SC_P3_LeakageTestA.AlarmTime.PT:= T#5s;
			SC_P3_LeakageTestA.IdleTime.IN:= TRUE;

			IF OpakovanyTest AND PocetOpakovaniTestu < 2 AND SC_P3_LeakageTestA.IdleTime.Q THEN
				SC_P3_LeakageTestA.ResetStep:= TRUE;
				SC_P3_LeakageTestA.Step:= 120;
			ELSIF OpakovanyTest AND PocetOpakovaniTestu >= 2 THEN
				PocetOpakovaniTestu:= 0;
				OpakovanyTest:= FALSE;
				SC_P3_LeakageTestA.ResetStep:= TRUE;
				SC_P3_LeakageTestA.Step:= 550;
			ELSIF NOT OpakovanyTest THEN
				PocetOpakovaniTestu:= 0;
				OpakovanyTest:= FALSE;
				SC_P3_LeakageTestA.ResetStep:= TRUE;
				SC_P3_LeakageTestA.Step:= 550;
			END_IF

			//**************************Odoslanie dát na server************************************//
		550:
			SC_P3_LeakageTestA.StepName:='550 - Automaticky Rezim - odoslanie stavu paletky na server';
			SC_P3_LeakageTestA.IdleTime.PT:= T#200ms;
			SC_P3_LeakageTestA.AlarmTime.PT:= T#5s;

			IF Linka.KOM_Panatrace_OFF THEN
				SC_P3_LeakageTestA.ResetStep:= TRUE;
				SC_P3_LeakageTestA.Step:= 560;
			ELSIF NOT SC_P3_LeakageTestA.Switch1 AND TRCB_P3_LeakageTestA_ST8A.STATUS.KOM_READY THEN
				TRCB_P3_LeakageTestA_ST8A.CMD.OdosliStavPaletky_TYP2:= TRUE;
				P3_LeakageTestA_Taktime.IN.START_MeraniaStratovehoCasu:= TRUE;
				SC_P3_LeakageTestA.Switch1:= TRUE;
			END_IF

			IF TRCB_P3_LeakageTestA_ST8A.STATUS.KomunikaciaUkoncena THEN
				TRCB_P3_LeakageTestA_ST8A.CMD.OdosliStavPaletky_TYP2:= FALSE;
				P3_LeakageTestA_Taktime.IN.START_MeraniaStratovehoCasu:= FALSE;
				SC_P3_LeakageTestA.ResetStep:= TRUE;
				SC_P3_LeakageTestA.Step:= 552;
			ELSIF TRCB_P3_LeakageTestA_ST8A.STATUS.KomunikaciaError THEN
				TRCB_P3_LeakageTestA_ST8A.CMD.OdosliStavPaletky_TYP2:= FALSE;
				P3_LeakageTestA_Taktime.IN.START_MeraniaStratovehoCasu:= FALSE;
				SC_P3_LeakageTestA.ResetStep:= TRUE;
				SC_P3_LeakageTestA.Step:= 557;
			END_IF

		552:
			SC_P3_LeakageTestA.StepName:='552 - Automaticky Rezim - kontrola odpovede servera';
			SC_P3_LeakageTestA.IdleTime.PT:= T#200ms;
			SC_P3_LeakageTestA.AlarmTime.PT:= T#5s;

			IF NOT TRCB_P3_LeakageTestA_ST8A.STATUS.KomunikaciaUkoncena THEN
				IF TRCB_P3_LeakageTestA_ST8A.OUTPUTS.PovolenieCinnostiNaPaletke = 'OK' THEN
					Paletka[i].STAV.Komunikacia_DONE:= TRUE;
					SC_P3_LeakageTestA.ResetStep:= TRUE;
					SC_P3_LeakageTestA.Step:= 560;
				ELSIF TRCB_P3_LeakageTestA_ST8A.OUTPUTS.PovolenieCinnostiNaPaletke = 'NG' THEN
					IF Paletka[i].STAV.StavPaletky <> 'TEST'THEN
						Paletka[i].STAV.StavPaletky:= 'NG';
					END_IF
					SC_P3_LeakageTestA.ResetStep:= TRUE;
					SC_P3_LeakageTestA.Step:= 560;
				END_IF
			END_IF

		555:
			SC_P3_LeakageTestA.StepName:='555 - Automaticky Rezim - vyziadanie stavu komunikacie zo serverom';
			SC_P3_LeakageTestA.IdleTime.PT:= T#200ms;
			SC_P3_LeakageTestA.AlarmTime.PT:= T#10s;

			IF NOT SC_P3_LeakageTestA.Switch1 AND TRCB_P3_LeakageTestA_ST8A.STATUS.KOM_READY THEN
				TRCB_P3_LeakageTestA_ST8A.CMD.VyziadajStavPanatrace_TYP4:= TRUE;
				SC_P3_LeakageTestA.Switch1:= TRUE;
			END_IF

			IF TRCB_P3_LeakageTestA_ST8A.STATUS.KomunikaciaUkoncena THEN
				TRCB_P3_LeakageTestA_ST8A.CMD.VyziadajStavPanatrace_TYP4:= FALSE;
				SC_P3_LeakageTestA.ResetStep:= TRUE;
				SC_P3_LeakageTestA.Step:= 556;
			ELSIF TRCB_P3_LeakageTestA_ST8A.STATUS.KomunikaciaError THEN
				TRCB_P3_LeakageTestA_ST8A.CMD.VyziadajStavPanatrace_TYP4:= FALSE;
				SC_P3_LeakageTestA.ResetStep:= TRUE;
				SC_P3_LeakageTestA.Step:= 557;
			END_IF

		556:
			SC_P3_LeakageTestA.StepName:='556 - Automaticky Rezim - kontrola odpovede servera';
			SC_P3_LeakageTestA.IdleTime.PT:= T#200ms;
			SC_P3_LeakageTestA.AlarmTime.PT:= T#5s;

			IF NOT TRCB_P3_LeakageTestA_ST8A.STATUS.KomunikaciaUkoncena THEN
				IF TRCB_P3_LeakageTestA_ST8A.OUTPUTS.DruhCinnostiNaPaletke = '0;Generating' THEN
					SC_P3_LeakageTestA.ResetStep:= TRUE;
					SC_P3_LeakageTestA.Step:= 557;
				ELSIF TRCB_P3_LeakageTestA_ST8A.OUTPUTS.DruhCinnostiNaPaletke = '1;Request' THEN
					SC_P3_LeakageTestA.ResetStep:= TRUE;
					SC_P3_LeakageTestA.Step:= 557;
				ELSIF TRCB_P3_LeakageTestA_ST8A.OUTPUTS.DruhCinnostiNaPaletke = '2;Report' THEN
					SC_P3_LeakageTestA.ResetStep:= TRUE;
					SC_P3_LeakageTestA.Step:= 550;
				ELSIF TRCB_P3_LeakageTestA_ST8A.OUTPUTS.DruhCinnostiNaPaletke = '3;Wedding' THEN
					SC_P3_LeakageTestA.ResetStep:= TRUE;
					SC_P3_LeakageTestA.Step:= 557;
				ELSIF TRCB_P3_LeakageTestA_ST8A.OUTPUTS.DruhCinnostiNaPaletke = '4;Status' THEN
					SC_P3_LeakageTestA.ResetStep:= TRUE;
					SC_P3_LeakageTestA.Step:= 557;
				ELSIF TRCB_P3_LeakageTestA_ST8A.OUTPUTS.DruhCinnostiNaPaletke = '5;' THEN
					SC_P3_LeakageTestA.ResetStep:= TRUE;
					SC_P3_LeakageTestA.Step:= 557;
				ELSE
					SC_P3_LeakageTestA.ResetStep:= TRUE;
					SC_P3_LeakageTestA.Step:= 557;
				END_IF
			END_IF

		557:
			SC_P3_LeakageTestA.StepName:='557 - Automaticky Rezim - rozhodnutie obsluhy po chybe komunikacie s Panatrace';
			SC_P3_LeakageTestA.IdleTime.PT:= T#200ms;
			SC_P3_LeakageTestA.AlarmTime.PT:= T#5s;

			P34_Vizu.ZobrazHL3_ST8:= TRUE;

			IF TRCB_P3_LeakTestA_OpatovnyDopyt THEN
				TRCB_P3_LeakTestA_OpatovnyDopyt:= FALSE;
				P34_Vizu.ZobrazHL3_ST8:= FALSE;
				SC_P3_LeakageTestA.ResetStep:= TRUE;
				SC_P3_LeakageTestA.Step:= 555;
			ELSIF TRCB_P3_LeakTestA_PaletkaNG THEN
				TRCB_P3_LeakTestA_PaletkaNG:= FALSE;
				P34_Vizu.ZobrazHL3_ST8:= FALSE;
				Paletka[i].STAV.StavPaletky := 'NG';
				SC_P3_LeakageTestA.ResetStep:= TRUE;
				SC_P3_LeakageTestA.Step:= 560;
			END_IF

			//***************************Vyvezenie paletky**********************************************//

		560:
			SC_P3_LeakageTestA.StepName:='560 - Automaticky Rezim - cakam na vyvezenie na zdvizku za leakage testom A';
			SC_P3_LeakageTestA.IdleTime.PT:= T#200ms;
			SC_P3_LeakageTestA.AlarmTime.PT:= T#5s;

			IF P3_LeakageTestA.KoniecCyklu THEN
				SC_P3_LeakageTestA.ResetStep:= TRUE;
				SC_P3_LeakageTestA.Step:= 0;
			ELSIF P3_Pracovisko.STAV.Porucha_ST5 THEN
				SC_P3_LeakageTestA.ResetStep:= TRUE;
				SC_P3_LeakageTestA.Step:= 0;
			ELSIF NOT P3_ZdvizkaZaLeakTestA.IN.PritomnostPaletky AND
				SC_P3_ZdvizkaZaLeakTestA.Step = 100 AND
				NOT P3_LeakageTestA.STAV.PrebiehaVyvezeniePaletky AND
				NOT P3_ZdvizkaZaLeakTestB.STAV.PrebiehaVyvezeniePaletkyNaTratA AND
				P3_ZdvizkaZaLeakTestA.IN.Zdvizka_StrednaPoloha AND
				P3_ZdvizkaZaLeakTestA.STAV.PoINIT AND
				P3_ZdvizkaZaLeakTestB.STAV.PoINIT THEN
				P3_LeakageTestA.OUT.ZasunStoper:= TRUE;
				P3_LeakageTestA.STAV.PrebiehaVyvezeniePaletky:= TRUE;
				SC_P3_LeakageTestA.ResetStep:= TRUE;
				SC_P3_LeakageTestA.Step:= 561;
			END_IF

		561:
			SC_P3_LeakageTestA.StepName:='561 - Automaticky Rezim - ukoncenie vyvazania na zdvizku za leakage testom A';
			SC_P3_LeakageTestA.IdleTime.PT:= T#200ms;
			SC_P3_LeakageTestA.AlarmTime.PT:= T#10s;

			SC_P3_LeakageTestA.IdleTime.IN:= NOT P3_LeakageTestA.RFID_hlava.PritomnostPaletky;
			SC_P3_LeakageTestA.AlarmTime.IN:= P3_LeakageTestA.RFID_hlava.PritomnostPaletky;

			IF NOT P3_LeakageTestA.RFID_hlava.PritomnostPaletky THEN
				P3_LeakageTestA.OUT.ZasunStoper:= FALSE;
				TestovaciKus:= FALSE;
				OpakovanyTest:= FALSE;
				PocetOpakovaniTestu:= 0;
				Paletka[i].PAR.StavPowerCP:= '';
				Paletka[i].STAV.Komunikacia_DONE:= FALSE;
				Reports.LeakageTest.CasPlnenia.StanicaA:= '';
				Reports.LeakageTest.VyslednyReport.StanicaA:= '';
				Reports.LeakageTest.CasStabilizacie.StanicaA:= '';
				Reports.LeakageTest.TlakPlnenia.StanicaA:= '';
				Reports.LeakageTest.ToleranciaPritlaku_MIN.StanicaA:= '';
				Reports.LeakageTest.ToleranciaPritlaku_MAX.StanicaA:= '';
				Reports.LeakageTest.TlakPritlaku.StanicaA:= '';
				Reports.LeakageTest.TlakUniku.StanicaA:= '';
				Reports.LeakageTest.Tolerancia.StanicaA:= '';
				SC_P3_LeakageTestA.ResetStep:= TRUE;
				SC_P3_LeakageTestA.Step:= 100;
			ELSIF SC_P3_LeakageTestA.AlarmTime.Q THEN
				P34_Alarmy[357]:= TRUE;
				P3_Pracovisko.STAV.Porucha_ST5:= TRUE;
			END_IF

			//*******************************************************Manuálny režim*******************************************************************************//
		700:
			SC_P3_LeakageTestA.StepName:='700 - Manualny Rezim';
			SC_P3_LeakageTestA.IdleTime.PT:= T#8s;
			SC_P3_LeakageTestA.AlarmTime.PT:= T#5s;

			//Vysunutie spodneho kopita//
			IF P3_LeakageTestA.CMD.RR_VysunSpodneKopito THEN
				P3_LeakageTestA.OUT.Kopito_ZASUN:= FALSE;
				P3_LeakageTestA.OUT.Kopito_VYSUN:= TRUE;
			ELSE
				P3_LeakageTestA.OUT.Kopito_VYSUN:= FALSE;
				P3_LeakageTestA.OUT.Kopito_ZASUN:= TRUE;
			END_IF

			//Testovacia sekvencia//
			IF P3_LeakageTestA.CMD.RR_TestovaciaSekvencia_START THEN
				IF P3_LeakageTestA.RFID_hlava.PritomnostPaletky THEN
					P3_LeakageTestA.STAV.RR_TestovaciaSekvencia_BUSY:= TRUE;
					SC_P3_LeakageTestA.ResetStep:= TRUE;
					SC_P3_LeakageTestA.Step:= 120;
				END_IF
				P3_LeakageTestA.CMD.RR_TestovaciaSekvencia_START:= FALSE;
			END_IF

			//Ovládanie centrovania paletky//
			IF P3_LeakageTestA.CMD.RR_VysunCentrovanie THEN
				P3_LeakageTestA.OUT.PneuZamokCentrovania_ODOMKNI:= TRUE;
				P3_LeakageTestA.OUT.Centrovanie_VYSUN:= TRUE;
			ELSE
				P3_LeakageTestA.OUT.PneuZamokCentrovania_ODOMKNI:= TRUE;
				P3_LeakageTestA.OUT.Centrovanie_VYSUN:= FALSE;
			END_IF

			//Ovládanie horného prítlaku//
			IF P3_LeakageTestA.CMD.RR_HornyPritlak_VYSUN THEN
				P3_LeakageTestA.OUT.PneuZamokZvonu_ODOMKNI:= TRUE;
				P3_LeakageTestA.OUT.HornyPritlak_ZASUN:= FALSE;
				P3_LeakageTestA.OUT.HornyPritlak_VYSUN:= TRUE;
				P3_LeakageTestA.CMD.RR_HornyPritlak_VYSUN:= FALSE;
			ELSIF P3_LeakageTestA.CMD.RR_HornyPritlak_ZASUN THEN
				P3_LeakageTestA.OUT.PneuZamokZvonu_ODOMKNI:= TRUE;
				P3_LeakageTestA.OUT.HornyPritlak_ZASUN:= TRUE;
				P3_LeakageTestA.OUT.HornyPritlak_VYSUN:= FALSE;
				P3_LeakageTestA.CMD.RR_HornyPritlak_ZASUN:= FALSE;
			END_IF

	END_CASE

END_PROGRAM

PROGRAM _EXIT
	(* Insert code here *)

END_PROGRAM
```

#### Variables.var - Local variables
```iecst
VAR
	SC_OvlCentrovacky : SequenceControlTyp;
	Centrovacku_VYSUN : BOOL;
	Centrovacku_ZASUN : BOOL;
	i : USINT;
	SC_OvlHornehoPritlaku : SequenceControlTyp := (0);
	HornyPritlak_VYSUN : BOOL := FALSE;
	HornyPritlak_ZASUN : BOOL := FALSE;
	CasPneniaREAL : REAL;
	CasStabilizacieREAL : REAL;
	TlakPlneniaREAL : REAL;
	ToleranciaREAL : REAL;
	TlakUnikuREAL : REAL;
	PocetDopytovNaServer : USINT := 0;
	PocetOpakovaniTestu : USINT := 0;
	TestovaciKus : BOOL := 0;
	OpakovanyTest : BOOL := 0;
	Triger_0 : BOOL := 0;
END_VAR
```

#### IOLinkKomunikacia.st
```iecst
ACTION IOLinkKomunikacia:

	//RFID snímač paletky//
	P3_LeakageTestA.RFID_hlava();

END_ACTION
```

#### OvlCentrovacky.st
```iecst
ACTION OvlCentrovacky:

	//Volanie funkcie SequenceControl//
	SequenceControl(SC:= SC_OvlCentrovacky);

	CASE SC_OvlCentrovacky.Step OF

		0:
			SC_OvlCentrovacky.StepName:= '0 - Nulovanie';
			Centrovacku_VYSUN:= FALSE;
			Centrovacku_ZASUN:= FALSE;

			IF SC_P3_LeakageTestA.Step <> 0 THEN
				SC_OvlCentrovacky.ResetStep:= TRUE;
				SC_OvlCentrovacky.Step:= 1;
			END_IF

		1:
			SC_OvlCentrovacky.StepName:= '1 - Rozhodnutie o cinnosti';
			IF Centrovacku_VYSUN THEN
				SC_OvlCentrovacky.Step:= 10;
			ELSIF Centrovacku_ZASUN THEN
				SC_OvlCentrovacky.Step:= 20;
			END_IF

		10:
			SC_OvlCentrovacky.StepName:= '10 - Vysunutie centrovacky';
			SC_OvlCentrovacky.IdleTime.PT:= T#3s;
			SC_OvlCentrovacky.AlarmTime.PT:= T#10s;

			IF P3_LeakageTestA.Automat THEN
				SC_OvlCentrovacky.AlarmTime.IN:= TRUE;
			ELSE
				SC_OvlCentrovacky.IdleTime.IN:= TRUE;
			END_IF

			IF NOT SC_OvlCentrovacky.Switch1 THEN
				P3_LeakageTestA.OUT.PneuZamokCentrovania_ODOMKNI:= TRUE;
                P3_LeakageTestA.OUT.Centrovanie_VYSUN:= TRUE;
				SC_OvlCentrovacky.Switch1:= TRUE;
			END_IF

			IF P3_LeakageTestA.IN.Centrovanie_VYSUNUTE OR SC_OvlCentrovacky.IdleTime.Q THEN
				SC_OvlCentrovacky.ResetStep:= TRUE;
				SC_OvlCentrovacky.Step:= 0;
			ELSIF SC_OvlCentrovacky.AlarmTime.Q THEN
				P34_Alarmy[302]:= TRUE;
				P3_Pracovisko.STAV.Porucha_ST5:= TRUE;
			END_IF

		20:
			SC_OvlCentrovacky.StepName:= '20 - Zasunutie centrovacky';
			SC_OvlCentrovacky.IdleTime.PT:= T#3s;
			SC_OvlCentrovacky.AlarmTime.PT:= T#10s;

			IF P3_LeakageTestA.Automat THEN
				SC_OvlCentrovacky.AlarmTime.IN:= TRUE;
			ELSE
				SC_OvlCentrovacky.IdleTime.IN:= TRUE;
			END_IF

			IF NOT SC_OvlCentrovacky.Switch1 THEN
				P3_LeakageTestA.OUT.Centrovanie_VYSUN:= FALSE;
                P3_LeakageTestA.OUT.PneuZamokCentrovania_ODOMKNI:= TRUE;
				SC_OvlCentrovacky.Switch1:= TRUE;
			END_IF

			IF P3_LeakageTestA.IN.Centrovanie_ZASUNUTE OR SC_OvlCentrovacky.IdleTime.Q THEN
				SC_OvlCentrovacky.ResetStep:= TRUE;
				SC_OvlCentrovacky.Step:= 0;
			ELSIF SC_OvlCentrovacky.AlarmTime.Q THEN
				P34_Alarmy[303]:= TRUE;
				P3_Pracovisko.STAV.Porucha_ST5:= TRUE;
			END_IF

	END_CASE

END_ACTION
```

#### OvlHornehoPritlaku.st
```iecst
ACTION OvlHornehoPritlaku:

	//Volanie funkcie SequenceControl//
	SequenceControl(SC:= SC_OvlHornehoPritlaku);

	CASE SC_OvlHornehoPritlaku.Step OF

		0:
			SC_OvlHornehoPritlaku.StepName:= '0 - Nulovanie';
			HornyPritlak_VYSUN:= FALSE;
			HornyPritlak_ZASUN:= FALSE;

			IF SC_P3_LeakageTestA.Step <> 0 THEN
				SC_OvlHornehoPritlaku.ResetStep:= TRUE;
				SC_OvlHornehoPritlaku.Step:= 1;
			END_IF

		1:
			SC_OvlHornehoPritlaku.StepName:= '1 - Rozhodnutie o cinnosti';
			IF HornyPritlak_VYSUN THEN
				SC_OvlHornehoPritlaku.Step:= 10;
			ELSIF HornyPritlak_ZASUN THEN
				SC_OvlHornehoPritlaku.Step:= 20;
			END_IF

		10:
			SC_OvlHornehoPritlaku.StepName:= '10 - Vysunutie horneho pritlaku';
			SC_OvlHornehoPritlaku.IdleTime.PT:= T#3s;
			SC_OvlHornehoPritlaku.AlarmTime.PT:= T#6s;

			IF P3_LeakageTestA.Automat THEN
				SC_OvlHornehoPritlaku.AlarmTime.IN:= TRUE;
			ELSE
				SC_OvlHornehoPritlaku.IdleTime.IN:= TRUE;
			END_IF

			IF NOT SC_OvlHornehoPritlaku.Switch1 THEN
				P3_LeakageTestA.OUT.PneuZamokZvonu_ODOMKNI:= TRUE;
				P3_LeakageTestA.OUT.HornyPritlak_ZASUN:= FALSE;
				P3_LeakageTestA.OUT.HornyPritlak_VYSUN:= TRUE;
				SC_OvlHornehoPritlaku.Switch1:= TRUE;
			END_IF

			IF P3_LeakageTestA.IN.HornyPritlak_VYSUNUTY OR SC_OvlHornehoPritlaku.IdleTime.Q THEN
				SC_OvlHornehoPritlaku.ResetStep:= TRUE;
				SC_OvlHornehoPritlaku.Step:= 0;
			ELSIF SC_OvlHornehoPritlaku.AlarmTime.Q THEN
				P34_Alarmy[306]:= TRUE;
				P3_Pracovisko.STAV.Porucha_ST5:= TRUE;
			END_IF

		20:
			SC_OvlHornehoPritlaku.StepName:= '20 - Zasunutie horneho pritlaku';
			SC_OvlHornehoPritlaku.IdleTime.PT:= T#3s;
			SC_OvlHornehoPritlaku.AlarmTime.PT:= T#6s;

			IF P3_LeakageTestA.Automat THEN
				SC_OvlHornehoPritlaku.AlarmTime.IN:= TRUE;
			ELSE
				SC_OvlHornehoPritlaku.IdleTime.IN:= TRUE;
			END_IF

			IF NOT SC_OvlHornehoPritlaku.Switch1 THEN
				P3_LeakageTestA.OUT.PneuZamokZvonu_ODOMKNI:= TRUE;
				P3_LeakageTestA.OUT.HornyPritlak_VYSUN:= FALSE;
				P3_LeakageTestA.OUT.HornyPritlak_ZASUN:= TRUE;
				SC_OvlHornehoPritlaku.Switch1:= TRUE;
			END_IF

			IF P3_LeakageTestA.IN.HornyPritlak_ZASUNUTY OR SC_OvlHornehoPritlaku.IdleTime.Q THEN
				SC_OvlHornehoPritlaku.ResetStep:= TRUE;
				SC_OvlHornehoPritlaku.Step:= 0;
			ELSIF SC_OvlHornehoPritlaku.AlarmTime.Q THEN
				P34_Alarmy[307]:= TRUE;
				P3_Pracovisko.STAV.Porucha_ST5:= TRUE;
			END_IF

	END_CASE

END_ACTION
```

#### COM_Tester.st
```iecst
ACTION COM_Tester:

	//Vstupy z Testera do PLC//
	AteqLeakageTester_A.Stav_RESET_DONE:= AteqLeakageTester_A.Profinet_PLC_INPUTS[1].0;
	AteqLeakageTester_A.Stav_START_DONE:= AteqLeakageTester_A.Profinet_PLC_INPUTS[1].1;
	AteqLeakageTester_A.Stav_ZmenaProgramu_DONE:= AteqLeakageTester_A.Profinet_PLC_INPUTS[1].3;
	AteqLeakageTester_A.Stav_CitanieParametrov_OK:= AteqLeakageTester_A.Profinet_PLC_INPUTS[1].5;

    AteqLeakageTester_A.Stav_CitanieParametrov_ERROR:= AteqLeakageTester_A.Profinet_PLC_INPUTS[3].5;

	AteqLeakageTester_A.CisloAktualnehoProgramu.0:= AteqLeakageTester_A.Profinet_PLC_INPUTS[7].0;
	AteqLeakageTester_A.CisloAktualnehoProgramu.1:= AteqLeakageTester_A.Profinet_PLC_INPUTS[7].1;
	AteqLeakageTester_A.CisloAktualnehoProgramu.2:= AteqLeakageTester_A.Profinet_PLC_INPUTS[7].2;
	AteqLeakageTester_A.CisloAktualnehoProgramu.3:= AteqLeakageTester_A.Profinet_PLC_INPUTS[7].3;
	AteqLeakageTester_A.CisloAktualnehoProgramu.4:= AteqLeakageTester_A.Profinet_PLC_INPUTS[7].4;
	AteqLeakageTester_A.CisloAktualnehoProgramu.5:= AteqLeakageTester_A.Profinet_PLC_INPUTS[7].5;
	AteqLeakageTester_A.CisloAktualnehoProgramu.6:= AteqLeakageTester_A.Profinet_PLC_INPUTS[7].6;
	AteqLeakageTester_A.CisloAktualnehoProgramu.7:= AteqLeakageTester_A.Profinet_PLC_INPUTS[7].7;

	AteqLeakageTester_A.CisloAktualnehoProgramu.8:= AteqLeakageTester_A.Profinet_PLC_INPUTS[8].0;
	AteqLeakageTester_A.CisloAktualnehoProgramu.9:= AteqLeakageTester_A.Profinet_PLC_INPUTS[8].1;
	AteqLeakageTester_A.CisloAktualnehoProgramu.10:= AteqLeakageTester_A.Profinet_PLC_INPUTS[8].2;
	AteqLeakageTester_A.CisloAktualnehoProgramu.11:= AteqLeakageTester_A.Profinet_PLC_INPUTS[8].3;
	AteqLeakageTester_A.CisloAktualnehoProgramu.12:= AteqLeakageTester_A.Profinet_PLC_INPUTS[8].4;
	AteqLeakageTester_A.CisloAktualnehoProgramu.13:= AteqLeakageTester_A.Profinet_PLC_INPUTS[8].5;
	AteqLeakageTester_A.CisloAktualnehoProgramu.14:= AteqLeakageTester_A.Profinet_PLC_INPUTS[8].6;
	AteqLeakageTester_A.CisloAktualnehoProgramu.15:= AteqLeakageTester_A.Profinet_PLC_INPUTS[8].7;

	AteqLeakageTester_A.VysledokTestovania_OK:= AteqLeakageTester_A.Profinet_PLC_INPUTS[13].0;
	AteqLeakageTester_A.VysledokTestovania_NG:= AteqLeakageTester_A.Profinet_PLC_INPUTS[13].1;
	AteqLeakageTester_A.Stav_ERROR:= AteqLeakageTester_A.Profinet_PLC_INPUTS[13].3;
	AteqLeakageTester_A.Stav_READY:= AteqLeakageTester_A.Profinet_PLC_INPUTS[13].5;

    AteqLeakageTester_A.ReadParameter_1.0:= AteqLeakageTester_A.Profinet_PLC_INPUTS[35].0;
    AteqLeakageTester_A.ReadParameter_1.1:= AteqLeakageTester_A.Profinet_PLC_INPUTS[35].1;
    AteqLeakageTester_A.ReadParameter_1.2:= AteqLeakageTester_A.Profinet_PLC_INPUTS[35].2;
    AteqLeakageTester_A.ReadParameter_1.3:= AteqLeakageTester_A.Profinet_PLC_INPUTS[35].3;
    AteqLeakageTester_A.ReadParameter_1.4:= AteqLeakageTester_A.Profinet_PLC_INPUTS[35].4;
    AteqLeakageTester_A.ReadParameter_1.5:= AteqLeakageTester_A.Profinet_PLC_INPUTS[35].5;
    AteqLeakageTester_A.ReadParameter_1.6:= AteqLeakageTester_A.Profinet_PLC_INPUTS[35].6;
    AteqLeakageTester_A.ReadParameter_1.7:= AteqLeakageTester_A.Profinet_PLC_INPUTS[35].7;
    AteqLeakageTester_A.ReadParameter_1.8:= AteqLeakageTester_A.Profinet_PLC_INPUTS[36].0;
    AteqLeakageTester_A.ReadParameter_1.9:= AteqLeakageTester_A.Profinet_PLC_INPUTS[36].1;
    AteqLeakageTester_A.ReadParameter_1.10:= AteqLeakageTester_A.Profinet_PLC_INPUTS[36].2;
    AteqLeakageTester_A.ReadParameter_1.11:= AteqLeakageTester_A.Profinet_PLC_INPUTS[36].3;
    AteqLeakageTester_A.ReadParameter_1.12:= AteqLeakageTester_A.Profinet_PLC_INPUTS[36].4;
    AteqLeakageTester_A.ReadParameter_1.13:= AteqLeakageTester_A.Profinet_PLC_INPUTS[36].5;
    AteqLeakageTester_A.ReadParameter_1.14:= AteqLeakageTester_A.Profinet_PLC_INPUTS[36].6;
    AteqLeakageTester_A.ReadParameter_1.15:= AteqLeakageTester_A.Profinet_PLC_INPUTS[36].7;

    AteqLeakageTester_A.ReadParameter_2.0:= AteqLeakageTester_A.Profinet_PLC_INPUTS[41].0;
    AteqLeakageTester_A.ReadParameter_2.1:= AteqLeakageTester_A.Profinet_PLC_INPUTS[41].1;
    AteqLeakageTester_A.ReadParameter_2.2:= AteqLeakageTester_A.Profinet_PLC_INPUTS[41].2;
    AteqLeakageTester_A.ReadParameter_2.3:= AteqLeakageTester_A.Profinet_PLC_INPUTS[41].3;
    AteqLeakageTester_A.ReadParameter_2.4:= AteqLeakageTester_A.Profinet_PLC_INPUTS[41].4;
    AteqLeakageTester_A.ReadParameter_2.5:= AteqLeakageTester_A.Profinet_PLC_INPUTS[41].5;
    AteqLeakageTester_A.ReadParameter_2.6:= AteqLeakageTester_A.Profinet_PLC_INPUTS[41].6;
    AteqLeakageTester_A.ReadParameter_2.7:= AteqLeakageTester_A.Profinet_PLC_INPUTS[41].7;
    AteqLeakageTester_A.ReadParameter_2.8:= AteqLeakageTester_A.Profinet_PLC_INPUTS[42].0;
    AteqLeakageTester_A.ReadParameter_2.9:= AteqLeakageTester_A.Profinet_PLC_INPUTS[42].1;
    AteqLeakageTester_A.ReadParameter_2.10:= AteqLeakageTester_A.Profinet_PLC_INPUTS[42].2;
    AteqLeakageTester_A.ReadParameter_2.11:= AteqLeakageTester_A.Profinet_PLC_INPUTS[42].3;
    AteqLeakageTester_A.ReadParameter_2.12:= AteqLeakageTester_A.Profinet_PLC_INPUTS[42].4;
    AteqLeakageTester_A.ReadParameter_2.13:= AteqLeakageTester_A.Profinet_PLC_INPUTS[42].5;
    AteqLeakageTester_A.ReadParameter_2.14:= AteqLeakageTester_A.Profinet_PLC_INPUTS[42].6;
    AteqLeakageTester_A.ReadParameter_2.15:= AteqLeakageTester_A.Profinet_PLC_INPUTS[42].7;

    AteqLeakageTester_A.ReadParameter_3.0:= AteqLeakageTester_A.Profinet_PLC_INPUTS[47].0;
    AteqLeakageTester_A.ReadParameter_3.1:= AteqLeakageTester_A.Profinet_PLC_INPUTS[47].1;
    AteqLeakageTester_A.ReadParameter_3.2:= AteqLeakageTester_A.Profinet_PLC_INPUTS[47].2;
    AteqLeakageTester_A.ReadParameter_3.3:= AteqLeakageTester_A.Profinet_PLC_INPUTS[47].3;
    AteqLeakageTester_A.ReadParameter_3.4:= AteqLeakageTester_A.Profinet_PLC_INPUTS[47].4;
    AteqLeakageTester_A.ReadParameter_3.5:= AteqLeakageTester_A.Profinet_PLC_INPUTS[47].5;
    AteqLeakageTester_A.ReadParameter_3.6:= AteqLeakageTester_A.Profinet_PLC_INPUTS[47].6;
    AteqLeakageTester_A.ReadParameter_3.7:= AteqLeakageTester_A.Profinet_PLC_INPUTS[47].7;
    AteqLeakageTester_A.ReadParameter_3.8:= AteqLeakageTester_A.Profinet_PLC_INPUTS[48].0;
    AteqLeakageTester_A.ReadParameter_3.9:= AteqLeakageTester_A.Profinet_PLC_INPUTS[48].1;
    AteqLeakageTester_A.ReadParameter_3.10:= AteqLeakageTester_A.Profinet_PLC_INPUTS[48].2;
    AteqLeakageTester_A.ReadParameter_3.11:= AteqLeakageTester_A.Profinet_PLC_INPUTS[48].3;
    AteqLeakageTester_A.ReadParameter_3.12:= AteqLeakageTester_A.Profinet_PLC_INPUTS[48].4;
    AteqLeakageTester_A.ReadParameter_3.13:= AteqLeakageTester_A.Profinet_PLC_INPUTS[48].5;
    AteqLeakageTester_A.ReadParameter_3.14:= AteqLeakageTester_A.Profinet_PLC_INPUTS[48].6;
    AteqLeakageTester_A.ReadParameter_3.15:= AteqLeakageTester_A.Profinet_PLC_INPUTS[48].7;

    AteqLeakageTester_A.ReadParameter_4.0:= AteqLeakageTester_A.Profinet_PLC_INPUTS[53].0;
    AteqLeakageTester_A.ReadParameter_4.1:= AteqLeakageTester_A.Profinet_PLC_INPUTS[53].1;
    AteqLeakageTester_A.ReadParameter_4.2:= AteqLeakageTester_A.Profinet_PLC_INPUTS[53].2;
    AteqLeakageTester_A.ReadParameter_4.3:= AteqLeakageTester_A.Profinet_PLC_INPUTS[53].3;
    AteqLeakageTester_A.ReadParameter_4.4:= AteqLeakageTester_A.Profinet_PLC_INPUTS[53].4;
    AteqLeakageTester_A.ReadParameter_4.5:= AteqLeakageTester_A.Profinet_PLC_INPUTS[53].5;
    AteqLeakageTester_A.ReadParameter_4.6:= AteqLeakageTester_A.Profinet_PLC_INPUTS[53].6;
    AteqLeakageTester_A.ReadParameter_4.7:= AteqLeakageTester_A.Profinet_PLC_INPUTS[53].7;
    AteqLeakageTester_A.ReadParameter_4.8:= AteqLeakageTester_A.Profinet_PLC_INPUTS[54].0;
    AteqLeakageTester_A.ReadParameter_4.9:= AteqLeakageTester_A.Profinet_PLC_INPUTS[54].1;
    AteqLeakageTester_A.ReadParameter_4.10:= AteqLeakageTester_A.Profinet_PLC_INPUTS[54].2;
    AteqLeakageTester_A.ReadParameter_4.11:= AteqLeakageTester_A.Profinet_PLC_INPUTS[54].3;
    AteqLeakageTester_A.ReadParameter_4.12:= AteqLeakageTester_A.Profinet_PLC_INPUTS[54].4;
    AteqLeakageTester_A.ReadParameter_4.13:= AteqLeakageTester_A.Profinet_PLC_INPUTS[54].5;
    AteqLeakageTester_A.ReadParameter_4.14:= AteqLeakageTester_A.Profinet_PLC_INPUTS[54].6;
    AteqLeakageTester_A.ReadParameter_4.15:= AteqLeakageTester_A.Profinet_PLC_INPUTS[54].7;

    AteqLeakageTester_A.ReadParameter_5.0:= AteqLeakageTester_A.Profinet_PLC_INPUTS[24].0;
    AteqLeakageTester_A.ReadParameter_5.1:= AteqLeakageTester_A.Profinet_PLC_INPUTS[24].1;
    AteqLeakageTester_A.ReadParameter_5.2:= AteqLeakageTester_A.Profinet_PLC_INPUTS[24].2;
    AteqLeakageTester_A.ReadParameter_5.3:= AteqLeakageTester_A.Profinet_PLC_INPUTS[24].3;
    AteqLeakageTester_A.ReadParameter_5.4:= AteqLeakageTester_A.Profinet_PLC_INPUTS[24].4;
    AteqLeakageTester_A.ReadParameter_5.5:= AteqLeakageTester_A.Profinet_PLC_INPUTS[24].5;
    AteqLeakageTester_A.ReadParameter_5.6:= AteqLeakageTester_A.Profinet_PLC_INPUTS[24].6;
    AteqLeakageTester_A.ReadParameter_5.7:= AteqLeakageTester_A.Profinet_PLC_INPUTS[24].7;
    AteqLeakageTester_A.ReadParameter_5.8:= AteqLeakageTester_A.Profinet_PLC_INPUTS[25].0;
    AteqLeakageTester_A.ReadParameter_5.9:= AteqLeakageTester_A.Profinet_PLC_INPUTS[25].1;
    AteqLeakageTester_A.ReadParameter_5.10:= AteqLeakageTester_A.Profinet_PLC_INPUTS[25].2;
    AteqLeakageTester_A.ReadParameter_5.11:= AteqLeakageTester_A.Profinet_PLC_INPUTS[25].3;
    AteqLeakageTester_A.ReadParameter_5.12:= AteqLeakageTester_A.Profinet_PLC_INPUTS[25].4;
    AteqLeakageTester_A.ReadParameter_5.13:= AteqLeakageTester_A.Profinet_PLC_INPUTS[25].5;
    AteqLeakageTester_A.ReadParameter_5.14:= AteqLeakageTester_A.Profinet_PLC_INPUTS[25].6;
    AteqLeakageTester_A.ReadParameter_5.15:= AteqLeakageTester_A.Profinet_PLC_INPUTS[25].7;
    AteqLeakageTester_A.ReadParameter_5.16:= AteqLeakageTester_A.Profinet_PLC_INPUTS[26].0;
    AteqLeakageTester_A.ReadParameter_5.17:= AteqLeakageTester_A.Profinet_PLC_INPUTS[26].1;
    AteqLeakageTester_A.ReadParameter_5.18:= AteqLeakageTester_A.Profinet_PLC_INPUTS[26].2;
    AteqLeakageTester_A.ReadParameter_5.19:= AteqLeakageTester_A.Profinet_PLC_INPUTS[26].3;
    AteqLeakageTester_A.ReadParameter_5.20:= AteqLeakageTester_A.Profinet_PLC_INPUTS[26].4;
    AteqLeakageTester_A.ReadParameter_5.21:= AteqLeakageTester_A.Profinet_PLC_INPUTS[26].5;
    AteqLeakageTester_A.ReadParameter_5.22:= AteqLeakageTester_A.Profinet_PLC_INPUTS[26].6;
    AteqLeakageTester_A.ReadParameter_5.23:= AteqLeakageTester_A.Profinet_PLC_INPUTS[26].7;
    AteqLeakageTester_A.ReadParameter_5.24:= AteqLeakageTester_A.Profinet_PLC_INPUTS[27].0;
    AteqLeakageTester_A.ReadParameter_5.25:= AteqLeakageTester_A.Profinet_PLC_INPUTS[27].1;
    AteqLeakageTester_A.ReadParameter_5.26:= AteqLeakageTester_A.Profinet_PLC_INPUTS[27].2;
    AteqLeakageTester_A.ReadParameter_5.27:= AteqLeakageTester_A.Profinet_PLC_INPUTS[27].3;
    AteqLeakageTester_A.ReadParameter_5.28:= AteqLeakageTester_A.Profinet_PLC_INPUTS[27].4;
    AteqLeakageTester_A.ReadParameter_5.29:= AteqLeakageTester_A.Profinet_PLC_INPUTS[27].5;
    AteqLeakageTester_A.ReadParameter_5.30:= AteqLeakageTester_A.Profinet_PLC_INPUTS[27].6;
    AteqLeakageTester_A.ReadParameter_5.31:= AteqLeakageTester_A.Profinet_PLC_INPUTS[27].7;

	//Vystupy z PLC do Testera//
	AteqLeakageTester_A.Profinet_PLC_OUTPUTS[1].0:= AteqLeakageTester_A.RESET_Vysledkov;
	AteqLeakageTester_A.Profinet_PLC_OUTPUTS[1].1:= AteqLeakageTester_A.START_Testovania;
	AteqLeakageTester_A.Profinet_PLC_OUTPUTS[1].3:= AteqLeakageTester_A.ZMEN_Program;
	AteqLeakageTester_A.Profinet_PLC_OUTPUTS[1].5:= AteqLeakageTester_A.CitajParametreTestera;

	AteqLeakageTester_A.Profinet_PLC_OUTPUTS[7].0:= AteqLeakageTester_A.CisloZadanehoProgramu.0;
	AteqLeakageTester_A.Profinet_PLC_OUTPUTS[7].1:= AteqLeakageTester_A.CisloZadanehoProgramu.1;
	AteqLeakageTester_A.Profinet_PLC_OUTPUTS[7].2:= AteqLeakageTester_A.CisloZadanehoProgramu.2;
	AteqLeakageTester_A.Profinet_PLC_OUTPUTS[7].3:= AteqLeakageTester_A.CisloZadanehoProgramu.3;
	AteqLeakageTester_A.Profinet_PLC_OUTPUTS[7].4:= AteqLeakageTester_A.CisloZadanehoProgramu.4;
	AteqLeakageTester_A.Profinet_PLC_OUTPUTS[7].5:= AteqLeakageTester_A.CisloZadanehoProgramu.5;
	AteqLeakageTester_A.Profinet_PLC_OUTPUTS[7].6:= AteqLeakageTester_A.CisloZadanehoProgramu.6;
	AteqLeakageTester_A.Profinet_PLC_OUTPUTS[7].7:= AteqLeakageTester_A.CisloZadanehoProgramu.7;

	AteqLeakageTester_A.Profinet_PLC_OUTPUTS[8].0:= AteqLeakageTester_A.CisloZadanehoProgramu.8;
	AteqLeakageTester_A.Profinet_PLC_OUTPUTS[8].1:= AteqLeakageTester_A.CisloZadanehoProgramu.9;
	AteqLeakageTester_A.Profinet_PLC_OUTPUTS[8].2:= AteqLeakageTester_A.CisloZadanehoProgramu.10;
	AteqLeakageTester_A.Profinet_PLC_OUTPUTS[8].3:= AteqLeakageTester_A.CisloZadanehoProgramu.11;
	AteqLeakageTester_A.Profinet_PLC_OUTPUTS[8].4:= AteqLeakageTester_A.CisloZadanehoProgramu.12;
	AteqLeakageTester_A.Profinet_PLC_OUTPUTS[8].5:= AteqLeakageTester_A.CisloZadanehoProgramu.13;
	AteqLeakageTester_A.Profinet_PLC_OUTPUTS[8].6:= AteqLeakageTester_A.CisloZadanehoProgramu.14;
	AteqLeakageTester_A.Profinet_PLC_OUTPUTS[8].7:= AteqLeakageTester_A.CisloZadanehoProgramu.15;

	AteqLeakageTester_A.PocetCitanychParametrov:= 4;
    AteqLeakageTester_A.IdentifikaciaParametra_1:= 1;
    AteqLeakageTester_A.IdentifikaciaParametra_2:= 2;
    AteqLeakageTester_A.IdentifikaciaParametra_3:= 66;
    AteqLeakageTester_A.IdentifikaciaParametra_4:= 60;

    //Vyčítané parametre//
    CasPneniaREAL:= UINT_TO_REAL(AteqLeakageTester_A.ReadParameter_1);
    AteqLeakageTester_A.CasPnenia:= CasPneniaREAL/1000;
    CasStabilizacieREAL:= UINT_TO_REAL(AteqLeakageTester_A.ReadParameter_2);
    AteqLeakageTester_A.CasStabilizacie:= CasStabilizacieREAL/1000;
    TlakPlneniaREAL:= UINT_TO_REAL(AteqLeakageTester_A.ReadParameter_3);
    AteqLeakageTester_A.TlakPlnenia:= TlakPlneniaREAL/1000;
    ToleranciaREAL:= UINT_TO_REAL(AteqLeakageTester_A.ReadParameter_4);
    AteqLeakageTester_A.Tolerancia:= ToleranciaREAL/1000;
    TlakUnikuREAL:= DINT_TO_REAL(AteqLeakageTester_A.ReadParameter_5);
    AteqLeakageTester_A.TlakUniku:= ((TlakUnikuREAL/1000)*6)/1536;

END_ACTION
```

### Program Logical/Program/Pracovisko_3/P3_LeakageTestB (IEC)
